// TIA Portal V20 export
FUNCTION_BLOCK "Sequence_20_Utility"   // FB240, LAD
AUTHOR : ERsystem_FA2_DH. Kim
// stored: IsIECCheckEnabled true, MemoryReserve 100, Namespace Unit1.Em6, SetENOAutomatically false
   VAR
      statSelectedJobNumber { ExternalWritable := 'False'} : DInt;   // Evaluated Job Number
      instSequenceLADStatus { ExternalWritable := 'False'} : "LAF_StatusLadSequence";
      instSequenceLADControl { ExternalWritable := 'False'} : "LAF_ControlLadSequence";
      statTonTime { ExternalAccessible := 'False'; ExternalVisible := 'False'; ExternalWritable := 'False'} : Array[0..999] of TON_TIME;
   END_VAR
   VAR CONSTANT
      STEP_IDLE : DInt := 1;
      STEP_IMMEDIATE_STOP : DInt := 9001;   // Step executed when an immediate stop command is triggered for the sequence (i.e. when unit is in state aborting)
      JOB_1_STEP_01 : DInt := 101;
      JOB_1_STEP_10 : DInt := 110;
      JOB_1_STEP_11 : DInt := 111;
      JOB_1_STEP_20 : DInt := 120;
      JOB_1_STEP_21 : DInt := 121;
      JOB_1_STEP_30 : DInt := 130;
      JOB_1_STEP_31 : DInt := 131;
      JOB_1_STEP_40 : DInt := 140;
      JOB_1_STEP_41 : DInt := 141;
      JOB_1_STEP_50 : DInt := 150;
      JOB_1_STEP_51 : DInt := 151;
      JOB_1_STEP_60 : DInt := 160;
      JOB_1_STEP_61 : DInt := 161;
      JOB_1_STEP_90 : DInt := 190;
      JOB_2_STEP_01 : DInt := 201;
      JOB_2_STEP_10 : DInt := 210;
      JOB_2_STEP_11 : DInt := 211;
      JOB_2_STEP_20 : DInt := 220;
      JOB_2_STEP_21 : DInt := 221;
      JOB_2_STEP_30 : DInt := 230;
      JOB_2_STEP_31 : DInt := 231;
      JOB_2_STEP_40 : DInt := 240;
      JOB_2_STEP_41 : DInt := 241;
      JOB_2_STEP_50 : DInt := 250;
      JOB_2_STEP_51 : DInt := 251;
      JOB_2_STEP_60 : DInt := 260;
      JOB_2_STEP_61 : DInt := 261;
      JOB_2_STEP_90 : DInt := 290;
   END_VAR
   VAR_TEMP   // added for the SCL form of the ladder/FBD networks
      _w1 : Bool;
   END_VAR
BEGIN

REGION Network 1: BLOCK INFO HEADER
   // (company) / (C) Copyright (year)
   // ---------------------------------------------------------------------------------
   // Title:                             (Title of this block)
   // Comment/Function: (that is implemented in the block)
   // Library/Family:           (that the source is dedicated to)
   // Author:                        (department / person in charge / contact)
   // Target System:          (test system with FW version)
   // Engineering:              TIA Portal (SW version)
   // Restrictions:               (OB types, etc.)
   // Requirements:           (hardware, technological package, etc.)
   // ---------------------------------------------------------------------------------
   // Change log table:
   // Version          | Date             | Signature      | Expert in charge  | Changes applied ------------------------|----------------------|-------------------------|--------------------------------|-----------------------
   // 001.000.000 | yyyy-mm-dd | 0x00000000 | (name of expert) | First released version
END_REGION

REGION Network 2: DESCRIPTION
   // This is a template block provided by the Automation Framework. It can be used to create an own project.
   // The Block Info Header is prepared to put in your own data.
   // Description of the block could be added here and the docu created by Code2Docu.
END_REGION

REGION Network 3: ********************* CONTROL *************************
END_REGION

REGION Network 4: Sequence Control
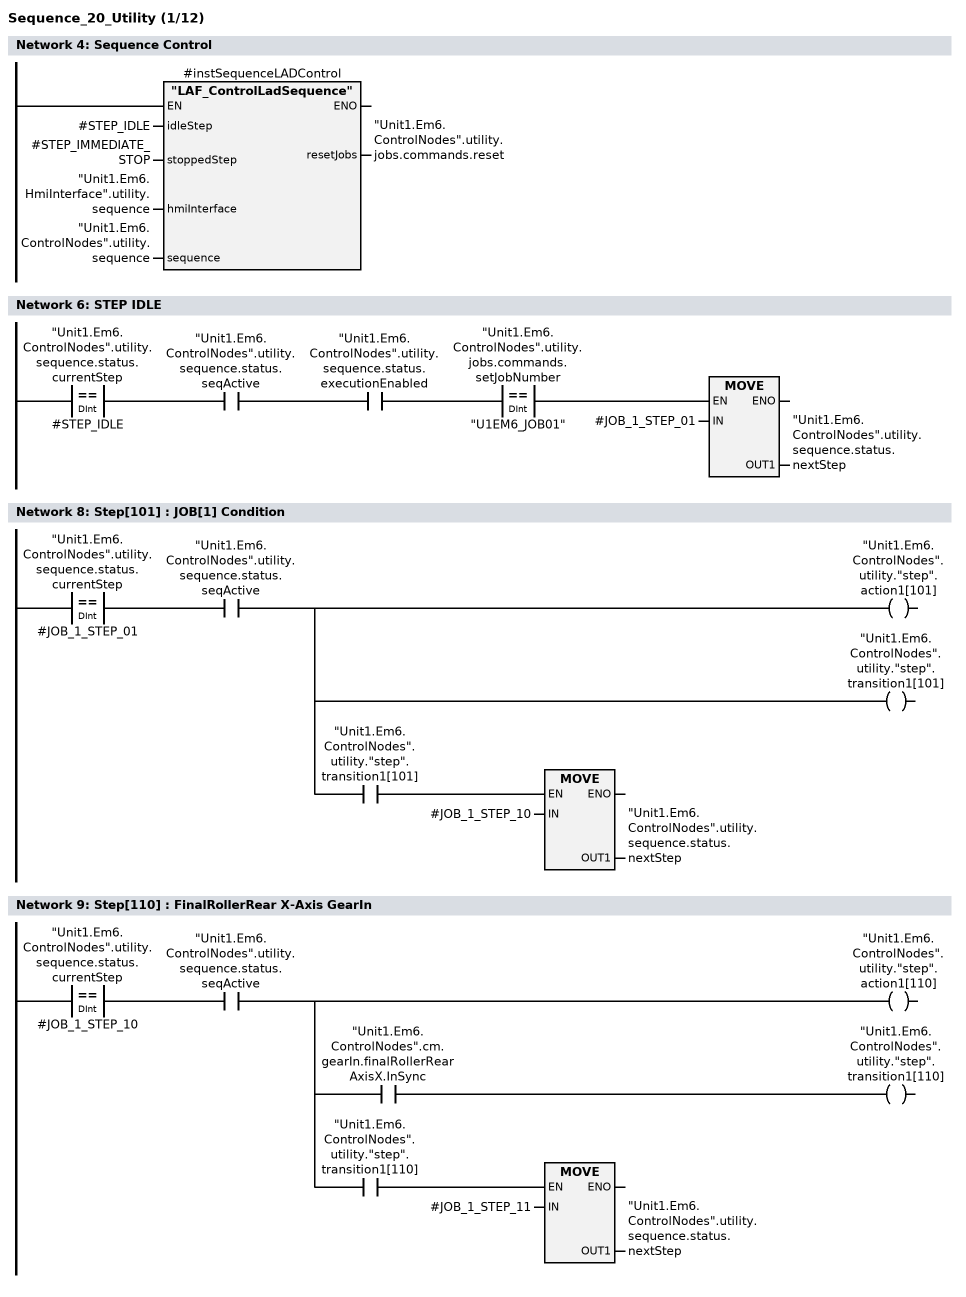
   RUNG wire#powerrail
      #instSequenceLADControl(idleStep := #STEP_IDLE, stoppedStep := #STEP_IMMEDIATE_STOP, hmiInterface := "Unit1.Em6.HmiInterface".utility.sequence, sequence := "Unit1.Em6.ControlNodes".utility.sequence, resetJobs => "Unit1.Em6.ControlNodes".utility.jobs.commands.reset)
   END_RUNG
   // the same network as SCL:
   #instSequenceLADControl(idleStep := #STEP_IDLE,   // "LAF_ControlLadSequence"
                           stoppedStep := #STEP_IMMEDIATE_STOP,
                           hmiInterface := "Unit1.Em6.HmiInterface".utility.sequence,
                           sequence := "Unit1.Em6.ControlNodes".utility.sequence,
                           resetJobs => "Unit1.Em6.ControlNodes".utility.jobs.commands.reset);
END_REGION

REGION Network 5: *************** JOB SELECT **************************
END_REGION

REGION Network 6: STEP IDLE
   RUNG wire#powerrail
      { S7_Templates := "SrcType := DInt" } EQ_Contact(in1 := "Unit1.Em6.ControlNodes".utility.sequence.status.currentStep, in2 := #STEP_IDLE)
      Contact( "Unit1.Em6.ControlNodes".utility.sequence.status.seqActive )
      Contact( "Unit1.Em6.ControlNodes".utility.sequence.status.executionEnabled )
      { S7_Templates := "SrcType := DInt" } EQ_Contact(in1 := "Unit1.Em6.ControlNodes".utility.jobs.commands.setJobNumber, in2 := "U1EM6_JOB01")
      Move(in := #JOB_1_STEP_01, out1 => "Unit1.Em6.ControlNodes".utility.sequence.status.nextStep)
   END_RUNG
   // the same network as SCL:
   IF ("Unit1.Em6.ControlNodes".utility.sequence.status.currentStep = #STEP_IDLE) AND "Unit1.Em6.ControlNodes".utility.sequence.status.seqActive AND "Unit1.Em6.ControlNodes".utility.sequence.status.executionEnabled AND ("Unit1.Em6.ControlNodes".utility.jobs.commands.setJobNumber = "U1EM6_JOB01") THEN
       "Unit1.Em6.ControlNodes".utility.sequence.status.nextStep := #JOB_1_STEP_01;
   END_IF;
END_REGION

REGION Network 7: *************** JOB[1] FinalRoller Gantry Home ************************
END_REGION

REGION Network 8: Step[101] : JOB[1] Condition
   RUNG wire#powerrail
      { S7_Templates := "SrcType := DInt" } EQ_Contact(in1 := "Unit1.Em6.ControlNodes".utility.sequence.status.currentStep, in2 := #JOB_1_STEP_01)
      Contact( "Unit1.Em6.ControlNodes".utility.sequence.status.seqActive )
      wire#w1
      Coil( "Unit1.Em6.ControlNodes".utility."step".action1[101] )
   END_RUNG
   RUNG wire#w1
      Coil( "Unit1.Em6.ControlNodes".utility."step".transition1[101] )
   END_RUNG
   RUNG wire#w1
      Contact( "Unit1.Em6.ControlNodes".utility."step".transition1[101] )
      Move(in := #JOB_1_STEP_10, out1 => "Unit1.Em6.ControlNodes".utility.sequence.status.nextStep)
   END_RUNG
   // the same network as SCL:
   "Unit1.Em6.ControlNodes".utility."step".action1[101] := ("Unit1.Em6.ControlNodes".utility.sequence.status.currentStep = #JOB_1_STEP_01) AND "Unit1.Em6.ControlNodes".utility.sequence.status.seqActive;
   "Unit1.Em6.ControlNodes".utility."step".transition1[101] := ("Unit1.Em6.ControlNodes".utility.sequence.status.currentStep = #JOB_1_STEP_01) AND "Unit1.Em6.ControlNodes".utility.sequence.status.seqActive;
   IF ("Unit1.Em6.ControlNodes".utility.sequence.status.currentStep = #JOB_1_STEP_01) AND "Unit1.Em6.ControlNodes".utility.sequence.status.seqActive AND "Unit1.Em6.ControlNodes".utility."step".transition1[101] THEN
       "Unit1.Em6.ControlNodes".utility.sequence.status.nextStep := #JOB_1_STEP_10;
   END_IF;
END_REGION

REGION Network 9: Step[110] : FinalRollerRear X-Axis GearIn
   RUNG wire#powerrail
      { S7_Templates := "SrcType := DInt" } EQ_Contact(in1 := "Unit1.Em6.ControlNodes".utility.sequence.status.currentStep, in2 := #JOB_1_STEP_10)
      Contact( "Unit1.Em6.ControlNodes".utility.sequence.status.seqActive )
      wire#w1
      Coil( "Unit1.Em6.ControlNodes".utility."step".action1[110] )
   END_RUNG
   RUNG wire#w1
      Contact( "Unit1.Em6.ControlNodes".cm.gearIn.finalRollerRearAxisX.InSync )
      Coil( "Unit1.Em6.ControlNodes".utility."step".transition1[110] )
   END_RUNG
   RUNG wire#w1
      Contact( "Unit1.Em6.ControlNodes".utility."step".transition1[110] )
      Move(in := #JOB_1_STEP_11, out1 => "Unit1.Em6.ControlNodes".utility.sequence.status.nextStep)
   END_RUNG
   // the same network as SCL:
   "Unit1.Em6.ControlNodes".utility."step".action1[110] := ("Unit1.Em6.ControlNodes".utility.sequence.status.currentStep = #JOB_1_STEP_10) AND "Unit1.Em6.ControlNodes".utility.sequence.status.seqActive;
   "Unit1.Em6.ControlNodes".utility."step".transition1[110] := ("Unit1.Em6.ControlNodes".utility.sequence.status.currentStep = #JOB_1_STEP_10) AND "Unit1.Em6.ControlNodes".utility.sequence.status.seqActive AND "Unit1.Em6.ControlNodes".cm.gearIn.finalRollerRearAxisX.InSync;
   IF ("Unit1.Em6.ControlNodes".utility.sequence.status.currentStep = #JOB_1_STEP_10) AND "Unit1.Em6.ControlNodes".utility.sequence.status.seqActive AND "Unit1.Em6.ControlNodes".utility."step".transition1[110] THEN
       "Unit1.Em6.ControlNodes".utility.sequence.status.nextStep := #JOB_1_STEP_11;
   END_IF;
END_REGION

REGION Network 10: Step[111] : FinalRollerRear X-Axis LimitSensor Off
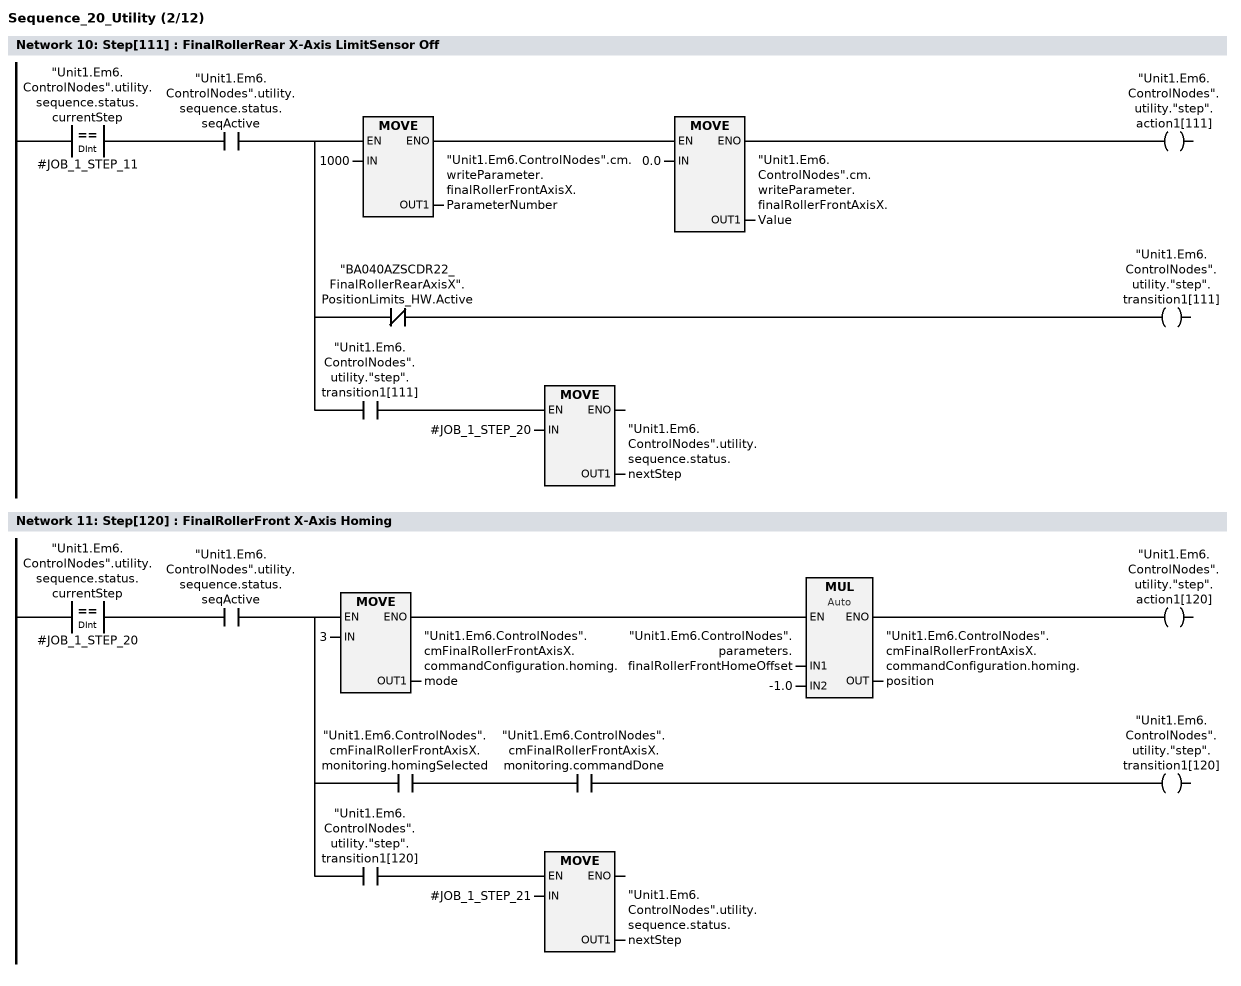
   RUNG wire#powerrail
      { S7_Templates := "SrcType := DInt" } EQ_Contact(in1 := "Unit1.Em6.ControlNodes".utility.sequence.status.currentStep, in2 := #JOB_1_STEP_11)
      Contact( "Unit1.Em6.ControlNodes".utility.sequence.status.seqActive )
      wire#w1
      Move(in := 1000, out1 => "Unit1.Em6.ControlNodes".cm.writeParameter.finalRollerFrontAxisX.ParameterNumber)
      Move(in := 0.0, out1 => "Unit1.Em6.ControlNodes".cm.writeParameter.finalRollerFrontAxisX.Value)
      Coil( "Unit1.Em6.ControlNodes".utility."step".action1[111] )
   END_RUNG
   RUNG wire#w1
      I_Contact( "BA040AZSCDR22_FinalRollerRearAxisX".PositionLimits_HW.Active )
      Coil( "Unit1.Em6.ControlNodes".utility."step".transition1[111] )
   END_RUNG
   RUNG wire#w1
      Contact( "Unit1.Em6.ControlNodes".utility."step".transition1[111] )
      Move(in := #JOB_1_STEP_20, out1 => "Unit1.Em6.ControlNodes".utility.sequence.status.nextStep)
   END_RUNG
   // the same network as SCL:
   #_w1 := ("Unit1.Em6.ControlNodes".utility.sequence.status.currentStep = #JOB_1_STEP_11) AND "Unit1.Em6.ControlNodes".utility.sequence.status.seqActive;
   IF #_w1 THEN
       "Unit1.Em6.ControlNodes".cm.writeParameter.finalRollerFrontAxisX.ParameterNumber := 1000;
       "Unit1.Em6.ControlNodes".cm.writeParameter.finalRollerFrontAxisX.Value := 0.0;
   END_IF;
   "Unit1.Em6.ControlNodes".utility."step".action1[111] := #_w1;
   "Unit1.Em6.ControlNodes".utility."step".transition1[111] := #_w1 AND NOT "BA040AZSCDR22_FinalRollerRearAxisX".PositionLimits_HW.Active;
   IF #_w1 AND "Unit1.Em6.ControlNodes".utility."step".transition1[111] THEN
       "Unit1.Em6.ControlNodes".utility.sequence.status.nextStep := #JOB_1_STEP_20;
   END_IF;
END_REGION

REGION Network 11: Step[120] : FinalRollerFront X-Axis Homing
   RUNG wire#powerrail
      { S7_Templates := "SrcType := DInt" } EQ_Contact(in1 := "Unit1.Em6.ControlNodes".utility.sequence.status.currentStep, in2 := #JOB_1_STEP_20)
      Contact( "Unit1.Em6.ControlNodes".utility.sequence.status.seqActive )
      wire#w1
      Move(in := 3, out1 => "Unit1.Em6.ControlNodes".cmFinalRollerFrontAxisX.commandConfiguration.homing.mode)
      Mul(in1 := "Unit1.Em6.ControlNodes".parameters.finalRollerFrontHomeOffset, in2 := -1.0, out => "Unit1.Em6.ControlNodes".cmFinalRollerFrontAxisX.commandConfiguration.homing.position)
      Coil( "Unit1.Em6.ControlNodes".utility."step".action1[120] )
   END_RUNG
   RUNG wire#w1
      Contact( "Unit1.Em6.ControlNodes".cmFinalRollerFrontAxisX.monitoring.homingSelected )
      Contact( "Unit1.Em6.ControlNodes".cmFinalRollerFrontAxisX.monitoring.commandDone )
      Coil( "Unit1.Em6.ControlNodes".utility."step".transition1[120] )
   END_RUNG
   RUNG wire#w1
      Contact( "Unit1.Em6.ControlNodes".utility."step".transition1[120] )
      Move(in := #JOB_1_STEP_21, out1 => "Unit1.Em6.ControlNodes".utility.sequence.status.nextStep)
   END_RUNG
   // the same network as SCL:
   #_w1 := ("Unit1.Em6.ControlNodes".utility.sequence.status.currentStep = #JOB_1_STEP_20) AND "Unit1.Em6.ControlNodes".utility.sequence.status.seqActive;
   IF #_w1 THEN
       "Unit1.Em6.ControlNodes".cmFinalRollerFrontAxisX.commandConfiguration.homing.mode := 3;
       "Unit1.Em6.ControlNodes".cmFinalRollerFrontAxisX.commandConfiguration.homing.position := "Unit1.Em6.ControlNodes".parameters.finalRollerFrontHomeOffset * (-1.0);
   END_IF;
   "Unit1.Em6.ControlNodes".utility."step".action1[120] := #_w1;
   "Unit1.Em6.ControlNodes".utility."step".transition1[120] := #_w1 AND "Unit1.Em6.ControlNodes".cmFinalRollerFrontAxisX.monitoring.homingSelected AND "Unit1.Em6.ControlNodes".cmFinalRollerFrontAxisX.monitoring.commandDone;
   IF #_w1 AND "Unit1.Em6.ControlNodes".utility."step".transition1[120] THEN
       "Unit1.Em6.ControlNodes".utility.sequence.status.nextStep := #JOB_1_STEP_21;
   END_IF;
END_REGION

REGION Network 12: Step[121] : FinalRollerFront X-Axis Move Home
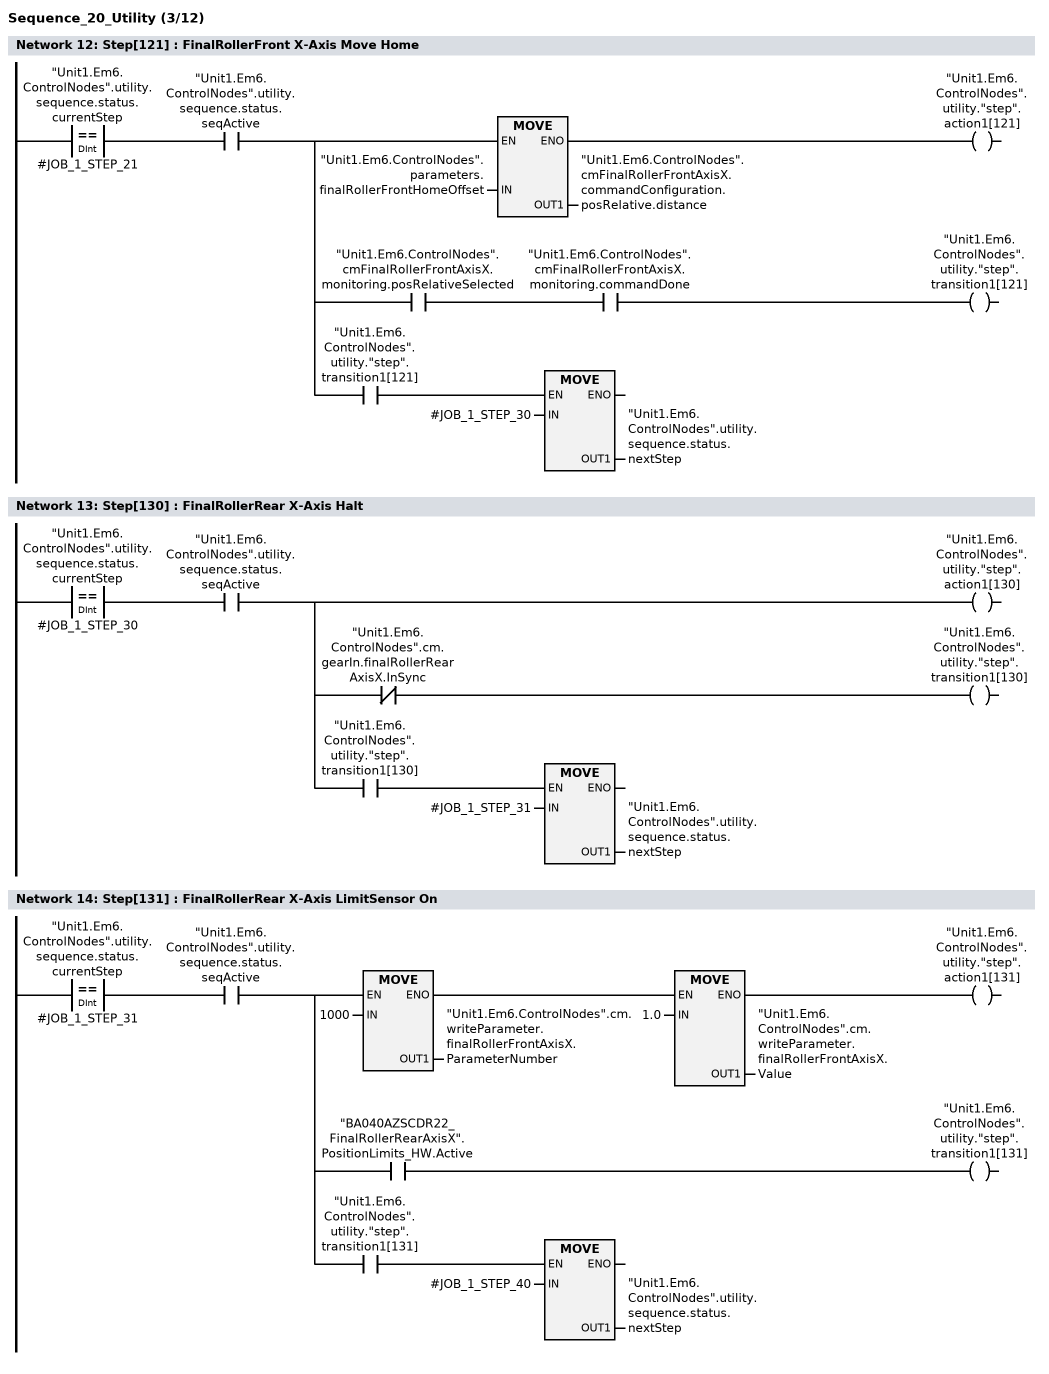
   RUNG wire#powerrail
      { S7_Templates := "SrcType := DInt" } EQ_Contact(in1 := "Unit1.Em6.ControlNodes".utility.sequence.status.currentStep, in2 := #JOB_1_STEP_21)
      Contact( "Unit1.Em6.ControlNodes".utility.sequence.status.seqActive )
      wire#w1
      Move(in := "Unit1.Em6.ControlNodes".parameters.finalRollerFrontHomeOffset, out1 => "Unit1.Em6.ControlNodes".cmFinalRollerFrontAxisX.commandConfiguration.posRelative.distance)
      Coil( "Unit1.Em6.ControlNodes".utility."step".action1[121] )
   END_RUNG
   RUNG wire#w1
      Contact( "Unit1.Em6.ControlNodes".cmFinalRollerFrontAxisX.monitoring.posRelativeSelected )
      Contact( "Unit1.Em6.ControlNodes".cmFinalRollerFrontAxisX.monitoring.commandDone )
      Coil( "Unit1.Em6.ControlNodes".utility."step".transition1[121] )
   END_RUNG
   RUNG wire#w1
      Contact( "Unit1.Em6.ControlNodes".utility."step".transition1[121] )
      Move(in := #JOB_1_STEP_30, out1 => "Unit1.Em6.ControlNodes".utility.sequence.status.nextStep)
   END_RUNG
   // the same network as SCL:
   #_w1 := ("Unit1.Em6.ControlNodes".utility.sequence.status.currentStep = #JOB_1_STEP_21) AND "Unit1.Em6.ControlNodes".utility.sequence.status.seqActive;
   IF #_w1 THEN
       "Unit1.Em6.ControlNodes".cmFinalRollerFrontAxisX.commandConfiguration.posRelative.distance := "Unit1.Em6.ControlNodes".parameters.finalRollerFrontHomeOffset;
   END_IF;
   "Unit1.Em6.ControlNodes".utility."step".action1[121] := #_w1;
   "Unit1.Em6.ControlNodes".utility."step".transition1[121] := #_w1 AND "Unit1.Em6.ControlNodes".cmFinalRollerFrontAxisX.monitoring.posRelativeSelected AND "Unit1.Em6.ControlNodes".cmFinalRollerFrontAxisX.monitoring.commandDone;
   IF #_w1 AND "Unit1.Em6.ControlNodes".utility."step".transition1[121] THEN
       "Unit1.Em6.ControlNodes".utility.sequence.status.nextStep := #JOB_1_STEP_30;
   END_IF;
END_REGION

REGION Network 13: Step[130] : FinalRollerRear X-Axis Halt
   RUNG wire#powerrail
      { S7_Templates := "SrcType := DInt" } EQ_Contact(in1 := "Unit1.Em6.ControlNodes".utility.sequence.status.currentStep, in2 := #JOB_1_STEP_30)
      Contact( "Unit1.Em6.ControlNodes".utility.sequence.status.seqActive )
      wire#w1
      Coil( "Unit1.Em6.ControlNodes".utility."step".action1[130] )
   END_RUNG
   RUNG wire#w1
      I_Contact( "Unit1.Em6.ControlNodes".cm.gearIn.finalRollerRearAxisX.InSync )
      Coil( "Unit1.Em6.ControlNodes".utility."step".transition1[130] )
   END_RUNG
   RUNG wire#w1
      Contact( "Unit1.Em6.ControlNodes".utility."step".transition1[130] )
      Move(in := #JOB_1_STEP_31, out1 => "Unit1.Em6.ControlNodes".utility.sequence.status.nextStep)
   END_RUNG
   // the same network as SCL:
   "Unit1.Em6.ControlNodes".utility."step".action1[130] := ("Unit1.Em6.ControlNodes".utility.sequence.status.currentStep = #JOB_1_STEP_30) AND "Unit1.Em6.ControlNodes".utility.sequence.status.seqActive;
   "Unit1.Em6.ControlNodes".utility."step".transition1[130] := ("Unit1.Em6.ControlNodes".utility.sequence.status.currentStep = #JOB_1_STEP_30) AND "Unit1.Em6.ControlNodes".utility.sequence.status.seqActive AND NOT "Unit1.Em6.ControlNodes".cm.gearIn.finalRollerRearAxisX.InSync;
   IF ("Unit1.Em6.ControlNodes".utility.sequence.status.currentStep = #JOB_1_STEP_30) AND "Unit1.Em6.ControlNodes".utility.sequence.status.seqActive AND "Unit1.Em6.ControlNodes".utility."step".transition1[130] THEN
       "Unit1.Em6.ControlNodes".utility.sequence.status.nextStep := #JOB_1_STEP_31;
   END_IF;
END_REGION

REGION Network 14: Step[131] : FinalRollerRear X-Axis LimitSensor On
   RUNG wire#powerrail
      { S7_Templates := "SrcType := DInt" } EQ_Contact(in1 := "Unit1.Em6.ControlNodes".utility.sequence.status.currentStep, in2 := #JOB_1_STEP_31)
      Contact( "Unit1.Em6.ControlNodes".utility.sequence.status.seqActive )
      wire#w1
      Move(in := 1000, out1 => "Unit1.Em6.ControlNodes".cm.writeParameter.finalRollerFrontAxisX.ParameterNumber)
      Move(in := 1.0, out1 => "Unit1.Em6.ControlNodes".cm.writeParameter.finalRollerFrontAxisX.Value)
      Coil( "Unit1.Em6.ControlNodes".utility."step".action1[131] )
   END_RUNG
   RUNG wire#w1
      Contact( "BA040AZSCDR22_FinalRollerRearAxisX".PositionLimits_HW.Active )
      Coil( "Unit1.Em6.ControlNodes".utility."step".transition1[131] )
   END_RUNG
   RUNG wire#w1
      Contact( "Unit1.Em6.ControlNodes".utility."step".transition1[131] )
      Move(in := #JOB_1_STEP_40, out1 => "Unit1.Em6.ControlNodes".utility.sequence.status.nextStep)
   END_RUNG
   // the same network as SCL:
   #_w1 := ("Unit1.Em6.ControlNodes".utility.sequence.status.currentStep = #JOB_1_STEP_31) AND "Unit1.Em6.ControlNodes".utility.sequence.status.seqActive;
   IF #_w1 THEN
       "Unit1.Em6.ControlNodes".cm.writeParameter.finalRollerFrontAxisX.ParameterNumber := 1000;
       "Unit1.Em6.ControlNodes".cm.writeParameter.finalRollerFrontAxisX.Value := 1.0;
   END_IF;
   "Unit1.Em6.ControlNodes".utility."step".action1[131] := #_w1;
   "Unit1.Em6.ControlNodes".utility."step".transition1[131] := #_w1 AND "BA040AZSCDR22_FinalRollerRearAxisX".PositionLimits_HW.Active;
   IF #_w1 AND "Unit1.Em6.ControlNodes".utility."step".transition1[131] THEN
       "Unit1.Em6.ControlNodes".utility.sequence.status.nextStep := #JOB_1_STEP_40;
   END_IF;
END_REGION

REGION Network 15: Step[140] : FinalRollerFront X-Axis GearIn
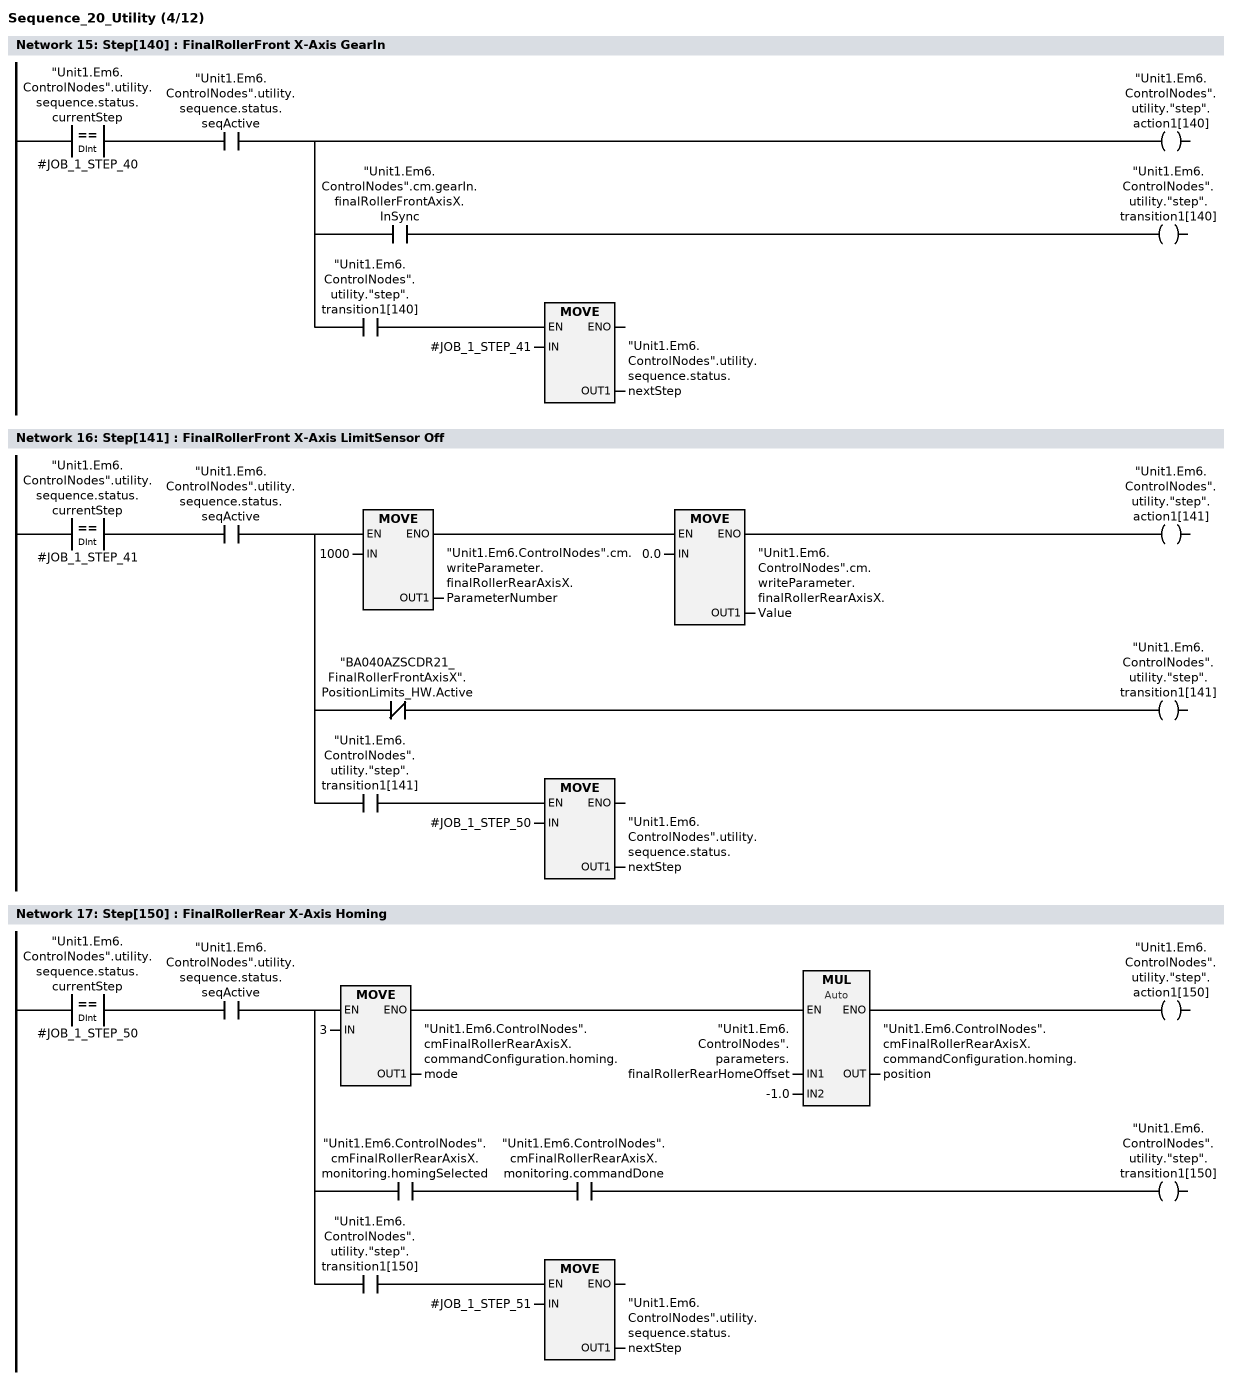
   RUNG wire#powerrail
      { S7_Templates := "SrcType := DInt" } EQ_Contact(in1 := "Unit1.Em6.ControlNodes".utility.sequence.status.currentStep, in2 := #JOB_1_STEP_40)
      Contact( "Unit1.Em6.ControlNodes".utility.sequence.status.seqActive )
      wire#w1
      Coil( "Unit1.Em6.ControlNodes".utility."step".action1[140] )
   END_RUNG
   RUNG wire#w1
      Contact( "Unit1.Em6.ControlNodes".cm.gearIn.finalRollerFrontAxisX.InSync )
      Coil( "Unit1.Em6.ControlNodes".utility."step".transition1[140] )
   END_RUNG
   RUNG wire#w1
      Contact( "Unit1.Em6.ControlNodes".utility."step".transition1[140] )
      Move(in := #JOB_1_STEP_41, out1 => "Unit1.Em6.ControlNodes".utility.sequence.status.nextStep)
   END_RUNG
   // the same network as SCL:
   "Unit1.Em6.ControlNodes".utility."step".action1[140] := ("Unit1.Em6.ControlNodes".utility.sequence.status.currentStep = #JOB_1_STEP_40) AND "Unit1.Em6.ControlNodes".utility.sequence.status.seqActive;
   "Unit1.Em6.ControlNodes".utility."step".transition1[140] := ("Unit1.Em6.ControlNodes".utility.sequence.status.currentStep = #JOB_1_STEP_40) AND "Unit1.Em6.ControlNodes".utility.sequence.status.seqActive AND "Unit1.Em6.ControlNodes".cm.gearIn.finalRollerFrontAxisX.InSync;
   IF ("Unit1.Em6.ControlNodes".utility.sequence.status.currentStep = #JOB_1_STEP_40) AND "Unit1.Em6.ControlNodes".utility.sequence.status.seqActive AND "Unit1.Em6.ControlNodes".utility."step".transition1[140] THEN
       "Unit1.Em6.ControlNodes".utility.sequence.status.nextStep := #JOB_1_STEP_41;
   END_IF;
END_REGION

REGION Network 16: Step[141] : FinalRollerFront X-Axis LimitSensor Off
   RUNG wire#powerrail
      { S7_Templates := "SrcType := DInt" } EQ_Contact(in1 := "Unit1.Em6.ControlNodes".utility.sequence.status.currentStep, in2 := #JOB_1_STEP_41)
      Contact( "Unit1.Em6.ControlNodes".utility.sequence.status.seqActive )
      wire#w1
      Move(in := 1000, out1 => "Unit1.Em6.ControlNodes".cm.writeParameter.finalRollerRearAxisX.ParameterNumber)
      Move(in := 0.0, out1 => "Unit1.Em6.ControlNodes".cm.writeParameter.finalRollerRearAxisX.Value)
      Coil( "Unit1.Em6.ControlNodes".utility."step".action1[141] )
   END_RUNG
   RUNG wire#w1
      I_Contact( "BA040AZSCDR21_FinalRollerFrontAxisX".PositionLimits_HW.Active )
      Coil( "Unit1.Em6.ControlNodes".utility."step".transition1[141] )
   END_RUNG
   RUNG wire#w1
      Contact( "Unit1.Em6.ControlNodes".utility."step".transition1[141] )
      Move(in := #JOB_1_STEP_50, out1 => "Unit1.Em6.ControlNodes".utility.sequence.status.nextStep)
   END_RUNG
   // the same network as SCL:
   #_w1 := ("Unit1.Em6.ControlNodes".utility.sequence.status.currentStep = #JOB_1_STEP_41) AND "Unit1.Em6.ControlNodes".utility.sequence.status.seqActive;
   IF #_w1 THEN
       "Unit1.Em6.ControlNodes".cm.writeParameter.finalRollerRearAxisX.ParameterNumber := 1000;
       "Unit1.Em6.ControlNodes".cm.writeParameter.finalRollerRearAxisX.Value := 0.0;
   END_IF;
   "Unit1.Em6.ControlNodes".utility."step".action1[141] := #_w1;
   "Unit1.Em6.ControlNodes".utility."step".transition1[141] := #_w1 AND NOT "BA040AZSCDR21_FinalRollerFrontAxisX".PositionLimits_HW.Active;
   IF #_w1 AND "Unit1.Em6.ControlNodes".utility."step".transition1[141] THEN
       "Unit1.Em6.ControlNodes".utility.sequence.status.nextStep := #JOB_1_STEP_50;
   END_IF;
END_REGION

REGION Network 17: Step[150] : FinalRollerRear X-Axis Homing
   RUNG wire#powerrail
      { S7_Templates := "SrcType := DInt" } EQ_Contact(in1 := "Unit1.Em6.ControlNodes".utility.sequence.status.currentStep, in2 := #JOB_1_STEP_50)
      Contact( "Unit1.Em6.ControlNodes".utility.sequence.status.seqActive )
      wire#w1
      Move(in := 3, out1 => "Unit1.Em6.ControlNodes".cmFinalRollerRearAxisX.commandConfiguration.homing.mode)
      Mul(in1 := "Unit1.Em6.ControlNodes".parameters.finalRollerRearHomeOffset, in2 := -1.0, out => "Unit1.Em6.ControlNodes".cmFinalRollerRearAxisX.commandConfiguration.homing.position)
      Coil( "Unit1.Em6.ControlNodes".utility."step".action1[150] )
   END_RUNG
   RUNG wire#w1
      Contact( "Unit1.Em6.ControlNodes".cmFinalRollerRearAxisX.monitoring.homingSelected )
      Contact( "Unit1.Em6.ControlNodes".cmFinalRollerRearAxisX.monitoring.commandDone )
      Coil( "Unit1.Em6.ControlNodes".utility."step".transition1[150] )
   END_RUNG
   RUNG wire#w1
      Contact( "Unit1.Em6.ControlNodes".utility."step".transition1[150] )
      Move(in := #JOB_1_STEP_51, out1 => "Unit1.Em6.ControlNodes".utility.sequence.status.nextStep)
   END_RUNG
   // the same network as SCL:
   #_w1 := ("Unit1.Em6.ControlNodes".utility.sequence.status.currentStep = #JOB_1_STEP_50) AND "Unit1.Em6.ControlNodes".utility.sequence.status.seqActive;
   IF #_w1 THEN
       "Unit1.Em6.ControlNodes".cmFinalRollerRearAxisX.commandConfiguration.homing.mode := 3;
       "Unit1.Em6.ControlNodes".cmFinalRollerRearAxisX.commandConfiguration.homing.position := "Unit1.Em6.ControlNodes".parameters.finalRollerRearHomeOffset * (-1.0);
   END_IF;
   "Unit1.Em6.ControlNodes".utility."step".action1[150] := #_w1;
   "Unit1.Em6.ControlNodes".utility."step".transition1[150] := #_w1 AND "Unit1.Em6.ControlNodes".cmFinalRollerRearAxisX.monitoring.homingSelected AND "Unit1.Em6.ControlNodes".cmFinalRollerRearAxisX.monitoring.commandDone;
   IF #_w1 AND "Unit1.Em6.ControlNodes".utility."step".transition1[150] THEN
       "Unit1.Em6.ControlNodes".utility.sequence.status.nextStep := #JOB_1_STEP_51;
   END_IF;
END_REGION

REGION Network 18: Step[151] : FinalRollerRear X-Axis Move Home
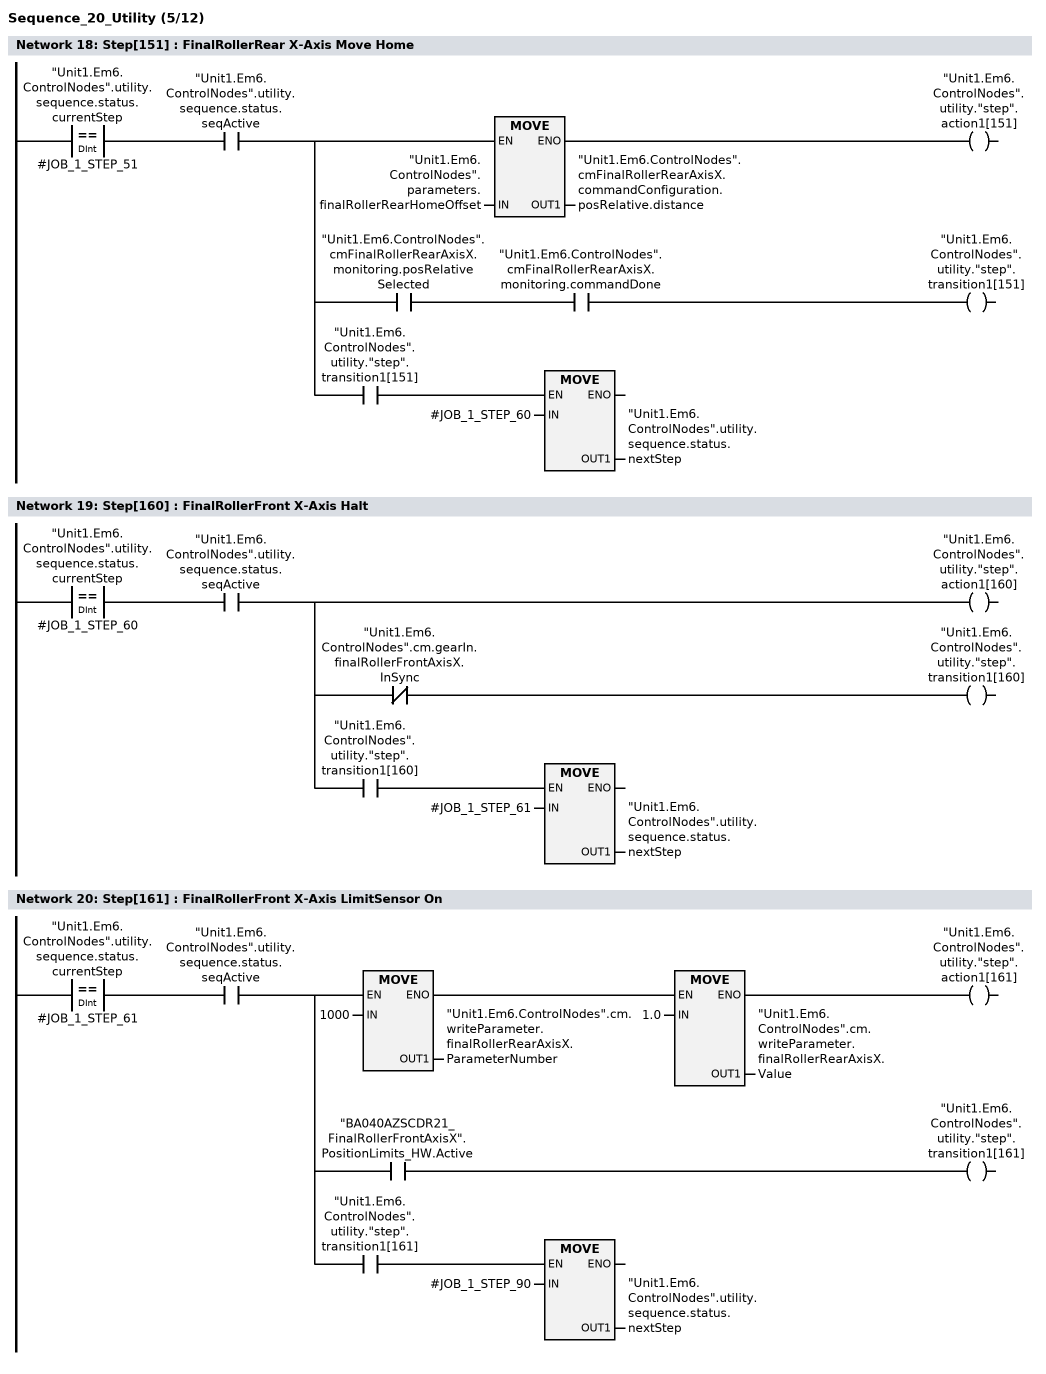
   RUNG wire#powerrail
      { S7_Templates := "SrcType := DInt" } EQ_Contact(in1 := "Unit1.Em6.ControlNodes".utility.sequence.status.currentStep, in2 := #JOB_1_STEP_51)
      Contact( "Unit1.Em6.ControlNodes".utility.sequence.status.seqActive )
      wire#w1
      Move(in := "Unit1.Em6.ControlNodes".parameters.finalRollerRearHomeOffset, out1 => "Unit1.Em6.ControlNodes".cmFinalRollerRearAxisX.commandConfiguration.posRelative.distance)
      Coil( "Unit1.Em6.ControlNodes".utility."step".action1[151] )
   END_RUNG
   RUNG wire#w1
      Contact( "Unit1.Em6.ControlNodes".cmFinalRollerRearAxisX.monitoring.posRelativeSelected )
      Contact( "Unit1.Em6.ControlNodes".cmFinalRollerRearAxisX.monitoring.commandDone )
      Coil( "Unit1.Em6.ControlNodes".utility."step".transition1[151] )
   END_RUNG
   RUNG wire#w1
      Contact( "Unit1.Em6.ControlNodes".utility."step".transition1[151] )
      Move(in := #JOB_1_STEP_60, out1 => "Unit1.Em6.ControlNodes".utility.sequence.status.nextStep)
   END_RUNG
   // the same network as SCL:
   #_w1 := ("Unit1.Em6.ControlNodes".utility.sequence.status.currentStep = #JOB_1_STEP_51) AND "Unit1.Em6.ControlNodes".utility.sequence.status.seqActive;
   IF #_w1 THEN
       "Unit1.Em6.ControlNodes".cmFinalRollerRearAxisX.commandConfiguration.posRelative.distance := "Unit1.Em6.ControlNodes".parameters.finalRollerRearHomeOffset;
   END_IF;
   "Unit1.Em6.ControlNodes".utility."step".action1[151] := #_w1;
   "Unit1.Em6.ControlNodes".utility."step".transition1[151] := #_w1 AND "Unit1.Em6.ControlNodes".cmFinalRollerRearAxisX.monitoring.posRelativeSelected AND "Unit1.Em6.ControlNodes".cmFinalRollerRearAxisX.monitoring.commandDone;
   IF #_w1 AND "Unit1.Em6.ControlNodes".utility."step".transition1[151] THEN
       "Unit1.Em6.ControlNodes".utility.sequence.status.nextStep := #JOB_1_STEP_60;
   END_IF;
END_REGION

REGION Network 19: Step[160] : FinalRollerFront X-Axis Halt
   RUNG wire#powerrail
      { S7_Templates := "SrcType := DInt" } EQ_Contact(in1 := "Unit1.Em6.ControlNodes".utility.sequence.status.currentStep, in2 := #JOB_1_STEP_60)
      Contact( "Unit1.Em6.ControlNodes".utility.sequence.status.seqActive )
      wire#w1
      Coil( "Unit1.Em6.ControlNodes".utility."step".action1[160] )
   END_RUNG
   RUNG wire#w1
      I_Contact( "Unit1.Em6.ControlNodes".cm.gearIn.finalRollerFrontAxisX.InSync )
      Coil( "Unit1.Em6.ControlNodes".utility."step".transition1[160] )
   END_RUNG
   RUNG wire#w1
      Contact( "Unit1.Em6.ControlNodes".utility."step".transition1[160] )
      Move(in := #JOB_1_STEP_61, out1 => "Unit1.Em6.ControlNodes".utility.sequence.status.nextStep)
   END_RUNG
   // the same network as SCL:
   "Unit1.Em6.ControlNodes".utility."step".action1[160] := ("Unit1.Em6.ControlNodes".utility.sequence.status.currentStep = #JOB_1_STEP_60) AND "Unit1.Em6.ControlNodes".utility.sequence.status.seqActive;
   "Unit1.Em6.ControlNodes".utility."step".transition1[160] := ("Unit1.Em6.ControlNodes".utility.sequence.status.currentStep = #JOB_1_STEP_60) AND "Unit1.Em6.ControlNodes".utility.sequence.status.seqActive AND NOT "Unit1.Em6.ControlNodes".cm.gearIn.finalRollerFrontAxisX.InSync;
   IF ("Unit1.Em6.ControlNodes".utility.sequence.status.currentStep = #JOB_1_STEP_60) AND "Unit1.Em6.ControlNodes".utility.sequence.status.seqActive AND "Unit1.Em6.ControlNodes".utility."step".transition1[160] THEN
       "Unit1.Em6.ControlNodes".utility.sequence.status.nextStep := #JOB_1_STEP_61;
   END_IF;
END_REGION

REGION Network 20: Step[161] : FinalRollerFront X-Axis LimitSensor On
   RUNG wire#powerrail
      { S7_Templates := "SrcType := DInt" } EQ_Contact(in1 := "Unit1.Em6.ControlNodes".utility.sequence.status.currentStep, in2 := #JOB_1_STEP_61)
      Contact( "Unit1.Em6.ControlNodes".utility.sequence.status.seqActive )
      wire#w1
      Move(in := 1000, out1 => "Unit1.Em6.ControlNodes".cm.writeParameter.finalRollerRearAxisX.ParameterNumber)
      Move(in := 1.0, out1 => "Unit1.Em6.ControlNodes".cm.writeParameter.finalRollerRearAxisX.Value)
      Coil( "Unit1.Em6.ControlNodes".utility."step".action1[161] )
   END_RUNG
   RUNG wire#w1
      Contact( "BA040AZSCDR21_FinalRollerFrontAxisX".PositionLimits_HW.Active )
      Coil( "Unit1.Em6.ControlNodes".utility."step".transition1[161] )
   END_RUNG
   RUNG wire#w1
      Contact( "Unit1.Em6.ControlNodes".utility."step".transition1[161] )
      Move(in := #JOB_1_STEP_90, out1 => "Unit1.Em6.ControlNodes".utility.sequence.status.nextStep)
   END_RUNG
   // the same network as SCL:
   #_w1 := ("Unit1.Em6.ControlNodes".utility.sequence.status.currentStep = #JOB_1_STEP_61) AND "Unit1.Em6.ControlNodes".utility.sequence.status.seqActive;
   IF #_w1 THEN
       "Unit1.Em6.ControlNodes".cm.writeParameter.finalRollerRearAxisX.ParameterNumber := 1000;
       "Unit1.Em6.ControlNodes".cm.writeParameter.finalRollerRearAxisX.Value := 1.0;
   END_IF;
   "Unit1.Em6.ControlNodes".utility."step".action1[161] := #_w1;
   "Unit1.Em6.ControlNodes".utility."step".transition1[161] := #_w1 AND "BA040AZSCDR21_FinalRollerFrontAxisX".PositionLimits_HW.Active;
   IF #_w1 AND "Unit1.Em6.ControlNodes".utility."step".transition1[161] THEN
       "Unit1.Em6.ControlNodes".utility.sequence.status.nextStep := #JOB_1_STEP_90;
   END_IF;
END_REGION

REGION Network 21: Step[190] : JOB[1] Step End
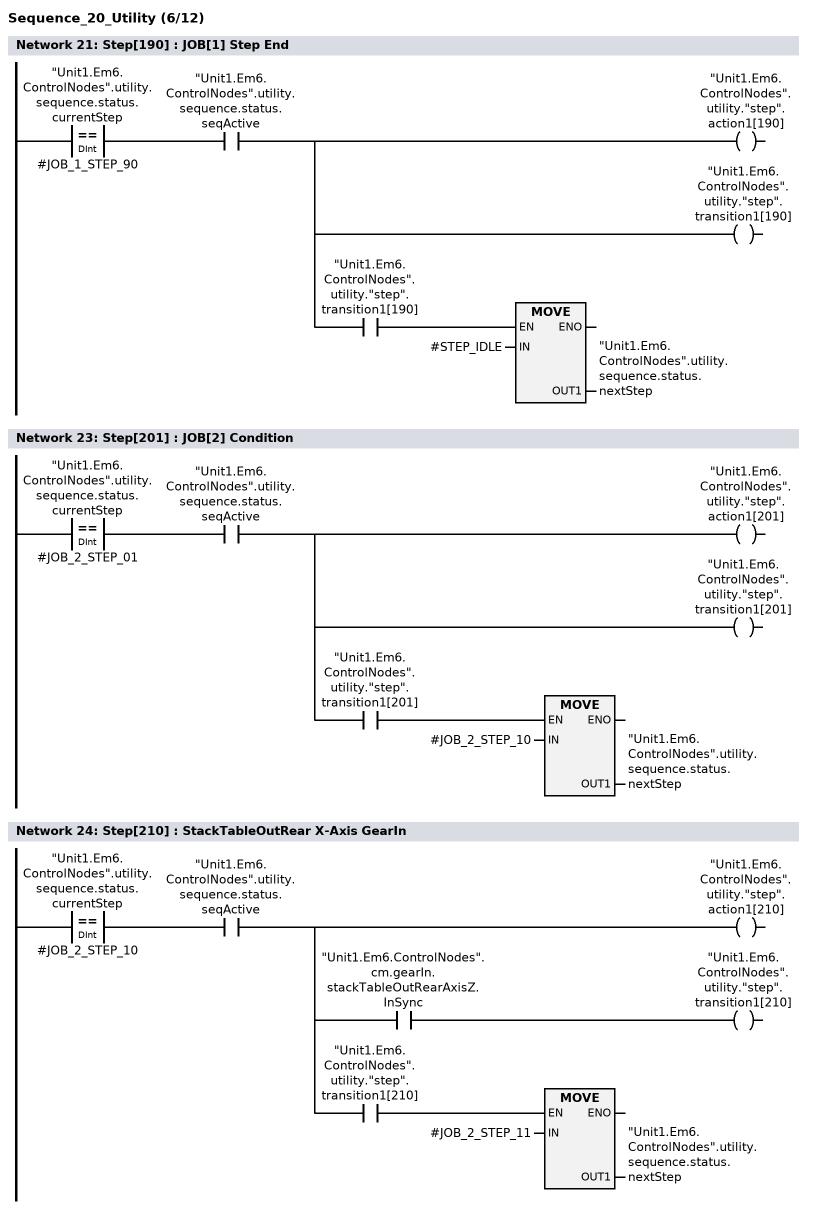
   RUNG wire#powerrail
      { S7_Templates := "SrcType := DInt" } EQ_Contact(in1 := "Unit1.Em6.ControlNodes".utility.sequence.status.currentStep, in2 := #JOB_1_STEP_90)
      Contact( "Unit1.Em6.ControlNodes".utility.sequence.status.seqActive )
      wire#w1
      Coil( "Unit1.Em6.ControlNodes".utility."step".action1[190] )
   END_RUNG
   RUNG wire#w1
      Coil( "Unit1.Em6.ControlNodes".utility."step".transition1[190] )
   END_RUNG
   RUNG wire#w1
      Contact( "Unit1.Em6.ControlNodes".utility."step".transition1[190] )
      Move(in := #STEP_IDLE, out1 => "Unit1.Em6.ControlNodes".utility.sequence.status.nextStep)
   END_RUNG
   // the same network as SCL:
   "Unit1.Em6.ControlNodes".utility."step".action1[190] := ("Unit1.Em6.ControlNodes".utility.sequence.status.currentStep = #JOB_1_STEP_90) AND "Unit1.Em6.ControlNodes".utility.sequence.status.seqActive;
   "Unit1.Em6.ControlNodes".utility."step".transition1[190] := ("Unit1.Em6.ControlNodes".utility.sequence.status.currentStep = #JOB_1_STEP_90) AND "Unit1.Em6.ControlNodes".utility.sequence.status.seqActive;
   IF ("Unit1.Em6.ControlNodes".utility.sequence.status.currentStep = #JOB_1_STEP_90) AND "Unit1.Em6.ControlNodes".utility.sequence.status.seqActive AND "Unit1.Em6.ControlNodes".utility."step".transition1[190] THEN
       "Unit1.Em6.ControlNodes".utility.sequence.status.nextStep := #STEP_IDLE;
   END_IF;
END_REGION

REGION Network 22: *************** JOB[2] StackTableOut Gantry Home ************************
END_REGION

REGION Network 23: Step[201] : JOB[2] Condition
   RUNG wire#powerrail
      { S7_Templates := "SrcType := DInt" } EQ_Contact(in1 := "Unit1.Em6.ControlNodes".utility.sequence.status.currentStep, in2 := #JOB_2_STEP_01)
      Contact( "Unit1.Em6.ControlNodes".utility.sequence.status.seqActive )
      wire#w1
      Coil( "Unit1.Em6.ControlNodes".utility."step".action1[201] )
   END_RUNG
   RUNG wire#w1
      Coil( "Unit1.Em6.ControlNodes".utility."step".transition1[201] )
   END_RUNG
   RUNG wire#w1
      Contact( "Unit1.Em6.ControlNodes".utility."step".transition1[201] )
      Move(in := #JOB_2_STEP_10, out1 => "Unit1.Em6.ControlNodes".utility.sequence.status.nextStep)
   END_RUNG
   // the same network as SCL:
   "Unit1.Em6.ControlNodes".utility."step".action1[201] := ("Unit1.Em6.ControlNodes".utility.sequence.status.currentStep = #JOB_2_STEP_01) AND "Unit1.Em6.ControlNodes".utility.sequence.status.seqActive;
   "Unit1.Em6.ControlNodes".utility."step".transition1[201] := ("Unit1.Em6.ControlNodes".utility.sequence.status.currentStep = #JOB_2_STEP_01) AND "Unit1.Em6.ControlNodes".utility.sequence.status.seqActive;
   IF ("Unit1.Em6.ControlNodes".utility.sequence.status.currentStep = #JOB_2_STEP_01) AND "Unit1.Em6.ControlNodes".utility.sequence.status.seqActive AND "Unit1.Em6.ControlNodes".utility."step".transition1[201] THEN
       "Unit1.Em6.ControlNodes".utility.sequence.status.nextStep := #JOB_2_STEP_10;
   END_IF;
END_REGION

REGION Network 24: Step[210] : StackTableOutRear X-Axis GearIn
   RUNG wire#powerrail
      { S7_Templates := "SrcType := DInt" } EQ_Contact(in1 := "Unit1.Em6.ControlNodes".utility.sequence.status.currentStep, in2 := #JOB_2_STEP_10)
      Contact( "Unit1.Em6.ControlNodes".utility.sequence.status.seqActive )
      wire#w1
      Coil( "Unit1.Em6.ControlNodes".utility."step".action1[210] )
   END_RUNG
   RUNG wire#w1
      Contact( "Unit1.Em6.ControlNodes".cm.gearIn.stackTableOutRearAxisZ.InSync )
      Coil( "Unit1.Em6.ControlNodes".utility."step".transition1[210] )
   END_RUNG
   RUNG wire#w1
      Contact( "Unit1.Em6.ControlNodes".utility."step".transition1[210] )
      Move(in := #JOB_2_STEP_11, out1 => "Unit1.Em6.ControlNodes".utility.sequence.status.nextStep)
   END_RUNG
   // the same network as SCL:
   "Unit1.Em6.ControlNodes".utility."step".action1[210] := ("Unit1.Em6.ControlNodes".utility.sequence.status.currentStep = #JOB_2_STEP_10) AND "Unit1.Em6.ControlNodes".utility.sequence.status.seqActive;
   "Unit1.Em6.ControlNodes".utility."step".transition1[210] := ("Unit1.Em6.ControlNodes".utility.sequence.status.currentStep = #JOB_2_STEP_10) AND "Unit1.Em6.ControlNodes".utility.sequence.status.seqActive AND "Unit1.Em6.ControlNodes".cm.gearIn.stackTableOutRearAxisZ.InSync;
   IF ("Unit1.Em6.ControlNodes".utility.sequence.status.currentStep = #JOB_2_STEP_10) AND "Unit1.Em6.ControlNodes".utility.sequence.status.seqActive AND "Unit1.Em6.ControlNodes".utility."step".transition1[210] THEN
       "Unit1.Em6.ControlNodes".utility.sequence.status.nextStep := #JOB_2_STEP_11;
   END_IF;
END_REGION

REGION Network 25: Step[211] : StackTableOutRear X-Axis LimitSensor Off
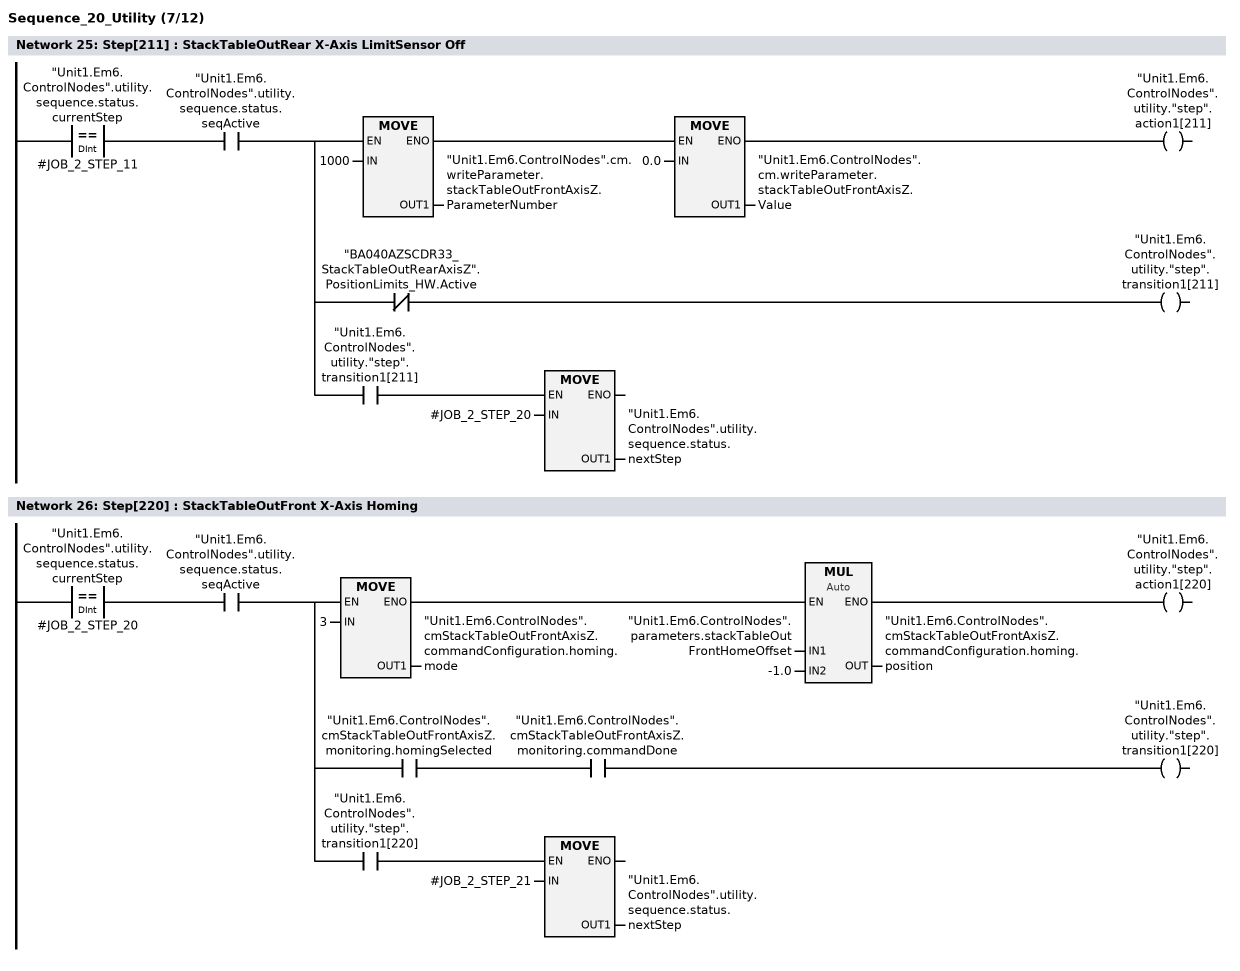
   RUNG wire#powerrail
      { S7_Templates := "SrcType := DInt" } EQ_Contact(in1 := "Unit1.Em6.ControlNodes".utility.sequence.status.currentStep, in2 := #JOB_2_STEP_11)
      Contact( "Unit1.Em6.ControlNodes".utility.sequence.status.seqActive )
      wire#w1
      Move(in := 1000, out1 => "Unit1.Em6.ControlNodes".cm.writeParameter.stackTableOutFrontAxisZ.ParameterNumber)
      Move(in := 0.0, out1 => "Unit1.Em6.ControlNodes".cm.writeParameter.stackTableOutFrontAxisZ.Value)
      Coil( "Unit1.Em6.ControlNodes".utility."step".action1[211] )
   END_RUNG
   RUNG wire#w1
      I_Contact( "BA040AZSCDR33_StackTableOutRearAxisZ".PositionLimits_HW.Active )
      Coil( "Unit1.Em6.ControlNodes".utility."step".transition1[211] )
   END_RUNG
   RUNG wire#w1
      Contact( "Unit1.Em6.ControlNodes".utility."step".transition1[211] )
      Move(in := #JOB_2_STEP_20, out1 => "Unit1.Em6.ControlNodes".utility.sequence.status.nextStep)
   END_RUNG
   // the same network as SCL:
   #_w1 := ("Unit1.Em6.ControlNodes".utility.sequence.status.currentStep = #JOB_2_STEP_11) AND "Unit1.Em6.ControlNodes".utility.sequence.status.seqActive;
   IF #_w1 THEN
       "Unit1.Em6.ControlNodes".cm.writeParameter.stackTableOutFrontAxisZ.ParameterNumber := 1000;
       "Unit1.Em6.ControlNodes".cm.writeParameter.stackTableOutFrontAxisZ.Value := 0.0;
   END_IF;
   "Unit1.Em6.ControlNodes".utility."step".action1[211] := #_w1;
   "Unit1.Em6.ControlNodes".utility."step".transition1[211] := #_w1 AND NOT "BA040AZSCDR33_StackTableOutRearAxisZ".PositionLimits_HW.Active;
   IF #_w1 AND "Unit1.Em6.ControlNodes".utility."step".transition1[211] THEN
       "Unit1.Em6.ControlNodes".utility.sequence.status.nextStep := #JOB_2_STEP_20;
   END_IF;
END_REGION

REGION Network 26: Step[220] : StackTableOutFront X-Axis Homing
   RUNG wire#powerrail
      { S7_Templates := "SrcType := DInt" } EQ_Contact(in1 := "Unit1.Em6.ControlNodes".utility.sequence.status.currentStep, in2 := #JOB_2_STEP_20)
      Contact( "Unit1.Em6.ControlNodes".utility.sequence.status.seqActive )
      wire#w1
      Move(in := 3, out1 => "Unit1.Em6.ControlNodes".cmStackTableOutFrontAxisZ.commandConfiguration.homing.mode)
      Mul(in1 := "Unit1.Em6.ControlNodes".parameters.stackTableOutFrontHomeOffset, in2 := -1.0, out => "Unit1.Em6.ControlNodes".cmStackTableOutFrontAxisZ.commandConfiguration.homing.position)
      Coil( "Unit1.Em6.ControlNodes".utility."step".action1[220] )
   END_RUNG
   RUNG wire#w1
      Contact( "Unit1.Em6.ControlNodes".cmStackTableOutFrontAxisZ.monitoring.homingSelected )
      Contact( "Unit1.Em6.ControlNodes".cmStackTableOutFrontAxisZ.monitoring.commandDone )
      Coil( "Unit1.Em6.ControlNodes".utility."step".transition1[220] )
   END_RUNG
   RUNG wire#w1
      Contact( "Unit1.Em6.ControlNodes".utility."step".transition1[220] )
      Move(in := #JOB_2_STEP_21, out1 => "Unit1.Em6.ControlNodes".utility.sequence.status.nextStep)
   END_RUNG
   // the same network as SCL:
   #_w1 := ("Unit1.Em6.ControlNodes".utility.sequence.status.currentStep = #JOB_2_STEP_20) AND "Unit1.Em6.ControlNodes".utility.sequence.status.seqActive;
   IF #_w1 THEN
       "Unit1.Em6.ControlNodes".cmStackTableOutFrontAxisZ.commandConfiguration.homing.mode := 3;
       "Unit1.Em6.ControlNodes".cmStackTableOutFrontAxisZ.commandConfiguration.homing.position := "Unit1.Em6.ControlNodes".parameters.stackTableOutFrontHomeOffset * (-1.0);
   END_IF;
   "Unit1.Em6.ControlNodes".utility."step".action1[220] := #_w1;
   "Unit1.Em6.ControlNodes".utility."step".transition1[220] := #_w1 AND "Unit1.Em6.ControlNodes".cmStackTableOutFrontAxisZ.monitoring.homingSelected AND "Unit1.Em6.ControlNodes".cmStackTableOutFrontAxisZ.monitoring.commandDone;
   IF #_w1 AND "Unit1.Em6.ControlNodes".utility."step".transition1[220] THEN
       "Unit1.Em6.ControlNodes".utility.sequence.status.nextStep := #JOB_2_STEP_21;
   END_IF;
END_REGION

REGION Network 27: Step[221] : StackTableOutFront X-Axis Move Home
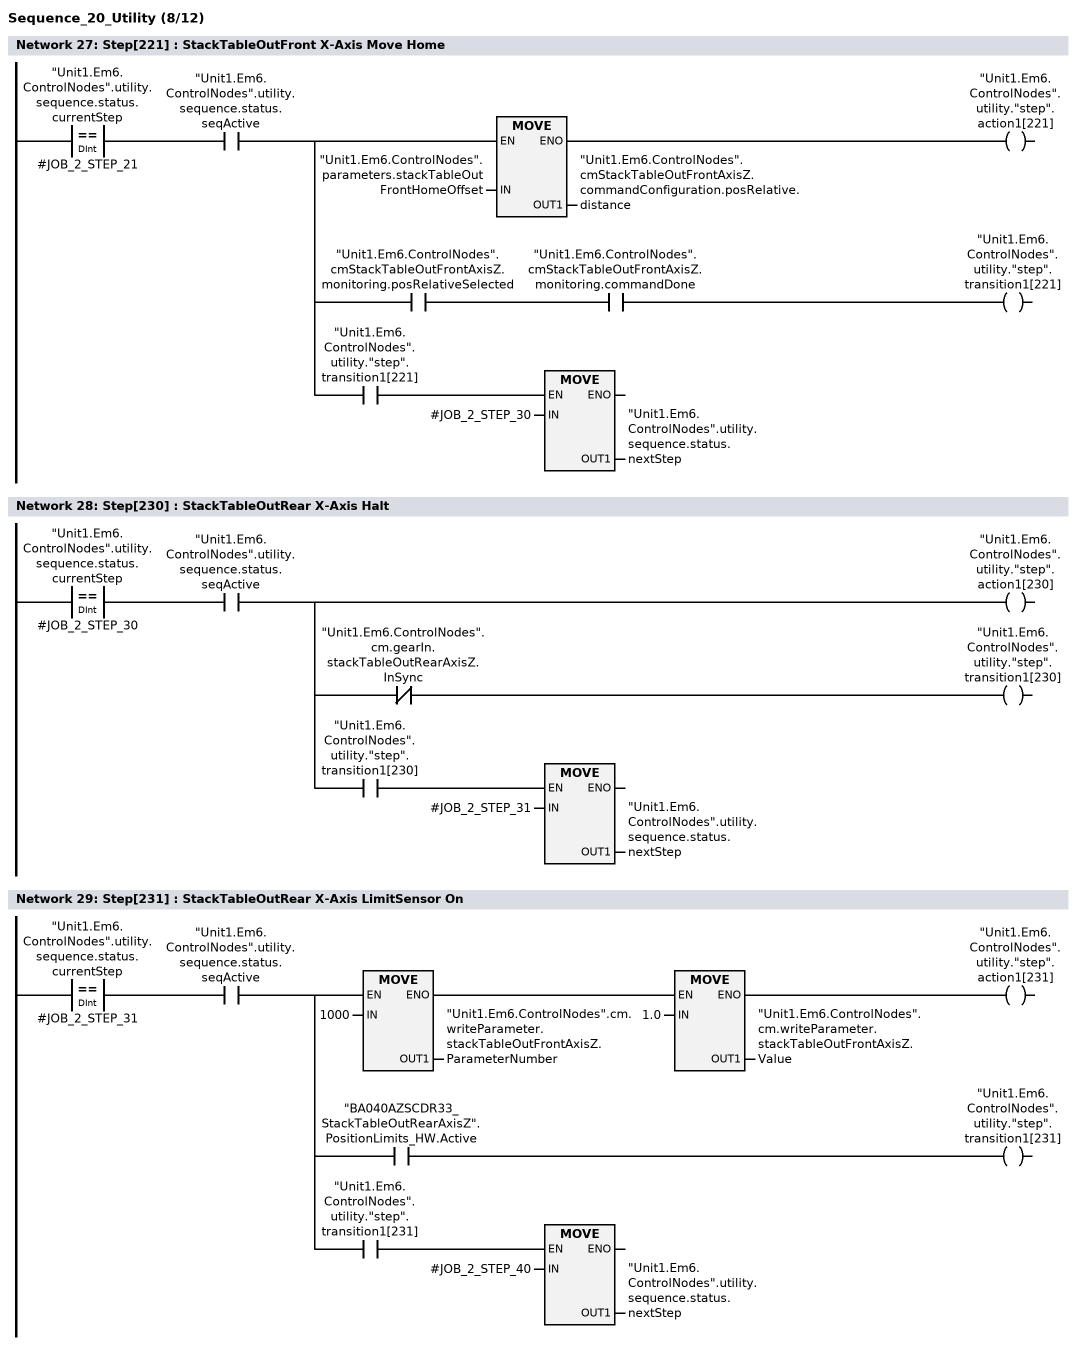
   RUNG wire#powerrail
      { S7_Templates := "SrcType := DInt" } EQ_Contact(in1 := "Unit1.Em6.ControlNodes".utility.sequence.status.currentStep, in2 := #JOB_2_STEP_21)
      Contact( "Unit1.Em6.ControlNodes".utility.sequence.status.seqActive )
      wire#w1
      Move(in := "Unit1.Em6.ControlNodes".parameters.stackTableOutFrontHomeOffset, out1 => "Unit1.Em6.ControlNodes".cmStackTableOutFrontAxisZ.commandConfiguration.posRelative.distance)
      Coil( "Unit1.Em6.ControlNodes".utility."step".action1[221] )
   END_RUNG
   RUNG wire#w1
      Contact( "Unit1.Em6.ControlNodes".cmStackTableOutFrontAxisZ.monitoring.posRelativeSelected )
      Contact( "Unit1.Em6.ControlNodes".cmStackTableOutFrontAxisZ.monitoring.commandDone )
      Coil( "Unit1.Em6.ControlNodes".utility."step".transition1[221] )
   END_RUNG
   RUNG wire#w1
      Contact( "Unit1.Em6.ControlNodes".utility."step".transition1[221] )
      Move(in := #JOB_2_STEP_30, out1 => "Unit1.Em6.ControlNodes".utility.sequence.status.nextStep)
   END_RUNG
   // the same network as SCL:
   #_w1 := ("Unit1.Em6.ControlNodes".utility.sequence.status.currentStep = #JOB_2_STEP_21) AND "Unit1.Em6.ControlNodes".utility.sequence.status.seqActive;
   IF #_w1 THEN
       "Unit1.Em6.ControlNodes".cmStackTableOutFrontAxisZ.commandConfiguration.posRelative.distance := "Unit1.Em6.ControlNodes".parameters.stackTableOutFrontHomeOffset;
   END_IF;
   "Unit1.Em6.ControlNodes".utility."step".action1[221] := #_w1;
   "Unit1.Em6.ControlNodes".utility."step".transition1[221] := #_w1 AND "Unit1.Em6.ControlNodes".cmStackTableOutFrontAxisZ.monitoring.posRelativeSelected AND "Unit1.Em6.ControlNodes".cmStackTableOutFrontAxisZ.monitoring.commandDone;
   IF #_w1 AND "Unit1.Em6.ControlNodes".utility."step".transition1[221] THEN
       "Unit1.Em6.ControlNodes".utility.sequence.status.nextStep := #JOB_2_STEP_30;
   END_IF;
END_REGION

REGION Network 28: Step[230] : StackTableOutRear X-Axis Halt
   RUNG wire#powerrail
      { S7_Templates := "SrcType := DInt" } EQ_Contact(in1 := "Unit1.Em6.ControlNodes".utility.sequence.status.currentStep, in2 := #JOB_2_STEP_30)
      Contact( "Unit1.Em6.ControlNodes".utility.sequence.status.seqActive )
      wire#w1
      Coil( "Unit1.Em6.ControlNodes".utility."step".action1[230] )
   END_RUNG
   RUNG wire#w1
      I_Contact( "Unit1.Em6.ControlNodes".cm.gearIn.stackTableOutRearAxisZ.InSync )
      Coil( "Unit1.Em6.ControlNodes".utility."step".transition1[230] )
   END_RUNG
   RUNG wire#w1
      Contact( "Unit1.Em6.ControlNodes".utility."step".transition1[230] )
      Move(in := #JOB_2_STEP_31, out1 => "Unit1.Em6.ControlNodes".utility.sequence.status.nextStep)
   END_RUNG
   // the same network as SCL:
   "Unit1.Em6.ControlNodes".utility."step".action1[230] := ("Unit1.Em6.ControlNodes".utility.sequence.status.currentStep = #JOB_2_STEP_30) AND "Unit1.Em6.ControlNodes".utility.sequence.status.seqActive;
   "Unit1.Em6.ControlNodes".utility."step".transition1[230] := ("Unit1.Em6.ControlNodes".utility.sequence.status.currentStep = #JOB_2_STEP_30) AND "Unit1.Em6.ControlNodes".utility.sequence.status.seqActive AND NOT "Unit1.Em6.ControlNodes".cm.gearIn.stackTableOutRearAxisZ.InSync;
   IF ("Unit1.Em6.ControlNodes".utility.sequence.status.currentStep = #JOB_2_STEP_30) AND "Unit1.Em6.ControlNodes".utility.sequence.status.seqActive AND "Unit1.Em6.ControlNodes".utility."step".transition1[230] THEN
       "Unit1.Em6.ControlNodes".utility.sequence.status.nextStep := #JOB_2_STEP_31;
   END_IF;
END_REGION

REGION Network 29: Step[231] : StackTableOutRear X-Axis LimitSensor On
   RUNG wire#powerrail
      { S7_Templates := "SrcType := DInt" } EQ_Contact(in1 := "Unit1.Em6.ControlNodes".utility.sequence.status.currentStep, in2 := #JOB_2_STEP_31)
      Contact( "Unit1.Em6.ControlNodes".utility.sequence.status.seqActive )
      wire#w1
      Move(in := 1000, out1 => "Unit1.Em6.ControlNodes".cm.writeParameter.stackTableOutFrontAxisZ.ParameterNumber)
      Move(in := 1.0, out1 => "Unit1.Em6.ControlNodes".cm.writeParameter.stackTableOutFrontAxisZ.Value)
      Coil( "Unit1.Em6.ControlNodes".utility."step".action1[231] )
   END_RUNG
   RUNG wire#w1
      Contact( "BA040AZSCDR33_StackTableOutRearAxisZ".PositionLimits_HW.Active )
      Coil( "Unit1.Em6.ControlNodes".utility."step".transition1[231] )
   END_RUNG
   RUNG wire#w1
      Contact( "Unit1.Em6.ControlNodes".utility."step".transition1[231] )
      Move(in := #JOB_2_STEP_40, out1 => "Unit1.Em6.ControlNodes".utility.sequence.status.nextStep)
   END_RUNG
   // the same network as SCL:
   #_w1 := ("Unit1.Em6.ControlNodes".utility.sequence.status.currentStep = #JOB_2_STEP_31) AND "Unit1.Em6.ControlNodes".utility.sequence.status.seqActive;
   IF #_w1 THEN
       "Unit1.Em6.ControlNodes".cm.writeParameter.stackTableOutFrontAxisZ.ParameterNumber := 1000;
       "Unit1.Em6.ControlNodes".cm.writeParameter.stackTableOutFrontAxisZ.Value := 1.0;
   END_IF;
   "Unit1.Em6.ControlNodes".utility."step".action1[231] := #_w1;
   "Unit1.Em6.ControlNodes".utility."step".transition1[231] := #_w1 AND "BA040AZSCDR33_StackTableOutRearAxisZ".PositionLimits_HW.Active;
   IF #_w1 AND "Unit1.Em6.ControlNodes".utility."step".transition1[231] THEN
       "Unit1.Em6.ControlNodes".utility.sequence.status.nextStep := #JOB_2_STEP_40;
   END_IF;
END_REGION

REGION Network 30: Step[240] : StackTableOutFront X-Axis GearIn
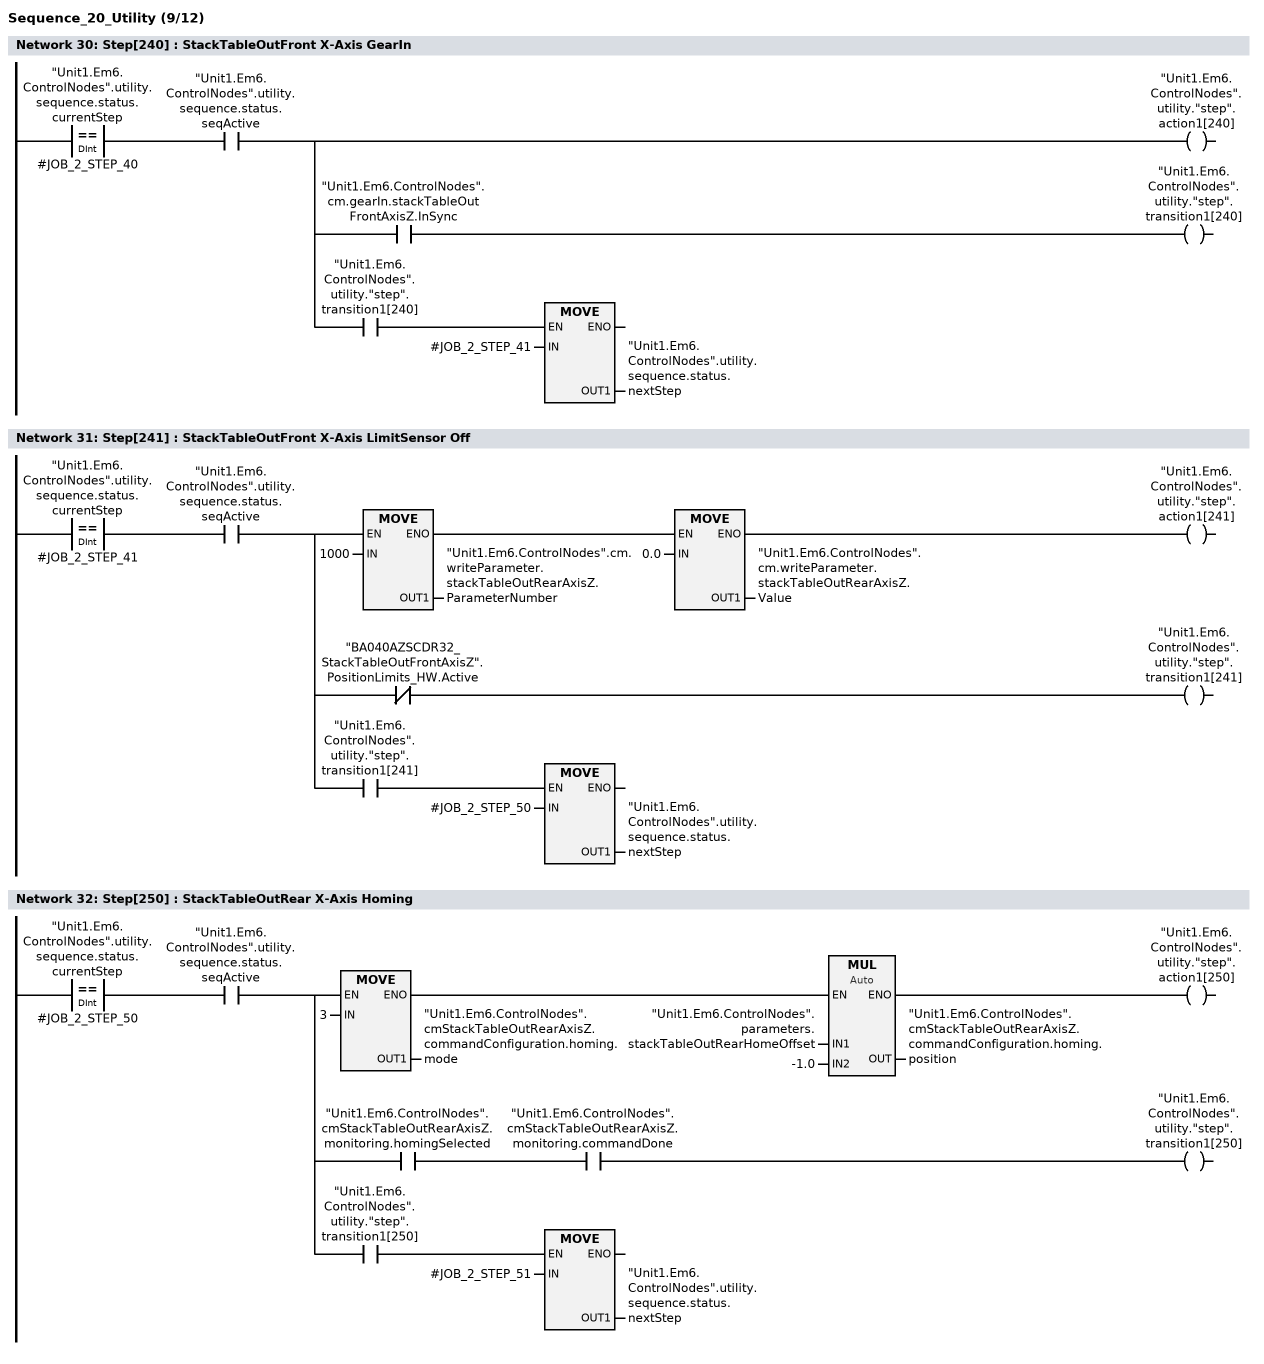
   RUNG wire#powerrail
      { S7_Templates := "SrcType := DInt" } EQ_Contact(in1 := "Unit1.Em6.ControlNodes".utility.sequence.status.currentStep, in2 := #JOB_2_STEP_40)
      Contact( "Unit1.Em6.ControlNodes".utility.sequence.status.seqActive )
      wire#w1
      Coil( "Unit1.Em6.ControlNodes".utility."step".action1[240] )
   END_RUNG
   RUNG wire#w1
      Contact( "Unit1.Em6.ControlNodes".cm.gearIn.stackTableOutFrontAxisZ.InSync )
      Coil( "Unit1.Em6.ControlNodes".utility."step".transition1[240] )
   END_RUNG
   RUNG wire#w1
      Contact( "Unit1.Em6.ControlNodes".utility."step".transition1[240] )
      Move(in := #JOB_2_STEP_41, out1 => "Unit1.Em6.ControlNodes".utility.sequence.status.nextStep)
   END_RUNG
   // the same network as SCL:
   "Unit1.Em6.ControlNodes".utility."step".action1[240] := ("Unit1.Em6.ControlNodes".utility.sequence.status.currentStep = #JOB_2_STEP_40) AND "Unit1.Em6.ControlNodes".utility.sequence.status.seqActive;
   "Unit1.Em6.ControlNodes".utility."step".transition1[240] := ("Unit1.Em6.ControlNodes".utility.sequence.status.currentStep = #JOB_2_STEP_40) AND "Unit1.Em6.ControlNodes".utility.sequence.status.seqActive AND "Unit1.Em6.ControlNodes".cm.gearIn.stackTableOutFrontAxisZ.InSync;
   IF ("Unit1.Em6.ControlNodes".utility.sequence.status.currentStep = #JOB_2_STEP_40) AND "Unit1.Em6.ControlNodes".utility.sequence.status.seqActive AND "Unit1.Em6.ControlNodes".utility."step".transition1[240] THEN
       "Unit1.Em6.ControlNodes".utility.sequence.status.nextStep := #JOB_2_STEP_41;
   END_IF;
END_REGION

REGION Network 31: Step[241] : StackTableOutFront X-Axis LimitSensor Off
   RUNG wire#powerrail
      { S7_Templates := "SrcType := DInt" } EQ_Contact(in1 := "Unit1.Em6.ControlNodes".utility.sequence.status.currentStep, in2 := #JOB_2_STEP_41)
      Contact( "Unit1.Em6.ControlNodes".utility.sequence.status.seqActive )
      wire#w1
      Move(in := 1000, out1 => "Unit1.Em6.ControlNodes".cm.writeParameter.stackTableOutRearAxisZ.ParameterNumber)
      Move(in := 0.0, out1 => "Unit1.Em6.ControlNodes".cm.writeParameter.stackTableOutRearAxisZ.Value)
      Coil( "Unit1.Em6.ControlNodes".utility."step".action1[241] )
   END_RUNG
   RUNG wire#w1
      I_Contact( "BA040AZSCDR32_StackTableOutFrontAxisZ".PositionLimits_HW.Active )
      Coil( "Unit1.Em6.ControlNodes".utility."step".transition1[241] )
   END_RUNG
   RUNG wire#w1
      Contact( "Unit1.Em6.ControlNodes".utility."step".transition1[241] )
      Move(in := #JOB_2_STEP_50, out1 => "Unit1.Em6.ControlNodes".utility.sequence.status.nextStep)
   END_RUNG
   // the same network as SCL:
   #_w1 := ("Unit1.Em6.ControlNodes".utility.sequence.status.currentStep = #JOB_2_STEP_41) AND "Unit1.Em6.ControlNodes".utility.sequence.status.seqActive;
   IF #_w1 THEN
       "Unit1.Em6.ControlNodes".cm.writeParameter.stackTableOutRearAxisZ.ParameterNumber := 1000;
       "Unit1.Em6.ControlNodes".cm.writeParameter.stackTableOutRearAxisZ.Value := 0.0;
   END_IF;
   "Unit1.Em6.ControlNodes".utility."step".action1[241] := #_w1;
   "Unit1.Em6.ControlNodes".utility."step".transition1[241] := #_w1 AND NOT "BA040AZSCDR32_StackTableOutFrontAxisZ".PositionLimits_HW.Active;
   IF #_w1 AND "Unit1.Em6.ControlNodes".utility."step".transition1[241] THEN
       "Unit1.Em6.ControlNodes".utility.sequence.status.nextStep := #JOB_2_STEP_50;
   END_IF;
END_REGION

REGION Network 32: Step[250] : StackTableOutRear X-Axis Homing
   RUNG wire#powerrail
      { S7_Templates := "SrcType := DInt" } EQ_Contact(in1 := "Unit1.Em6.ControlNodes".utility.sequence.status.currentStep, in2 := #JOB_2_STEP_50)
      Contact( "Unit1.Em6.ControlNodes".utility.sequence.status.seqActive )
      wire#w1
      Move(in := 3, out1 => "Unit1.Em6.ControlNodes".cmStackTableOutRearAxisZ.commandConfiguration.homing.mode)
      Mul(in1 := "Unit1.Em6.ControlNodes".parameters.stackTableOutRearHomeOffset, in2 := -1.0, out => "Unit1.Em6.ControlNodes".cmStackTableOutRearAxisZ.commandConfiguration.homing.position)
      Coil( "Unit1.Em6.ControlNodes".utility."step".action1[250] )
   END_RUNG
   RUNG wire#w1
      Contact( "Unit1.Em6.ControlNodes".cmStackTableOutRearAxisZ.monitoring.homingSelected )
      Contact( "Unit1.Em6.ControlNodes".cmStackTableOutRearAxisZ.monitoring.commandDone )
      Coil( "Unit1.Em6.ControlNodes".utility."step".transition1[250] )
   END_RUNG
   RUNG wire#w1
      Contact( "Unit1.Em6.ControlNodes".utility."step".transition1[250] )
      Move(in := #JOB_2_STEP_51, out1 => "Unit1.Em6.ControlNodes".utility.sequence.status.nextStep)
   END_RUNG
   // the same network as SCL:
   #_w1 := ("Unit1.Em6.ControlNodes".utility.sequence.status.currentStep = #JOB_2_STEP_50) AND "Unit1.Em6.ControlNodes".utility.sequence.status.seqActive;
   IF #_w1 THEN
       "Unit1.Em6.ControlNodes".cmStackTableOutRearAxisZ.commandConfiguration.homing.mode := 3;
       "Unit1.Em6.ControlNodes".cmStackTableOutRearAxisZ.commandConfiguration.homing.position := "Unit1.Em6.ControlNodes".parameters.stackTableOutRearHomeOffset * (-1.0);
   END_IF;
   "Unit1.Em6.ControlNodes".utility."step".action1[250] := #_w1;
   "Unit1.Em6.ControlNodes".utility."step".transition1[250] := #_w1 AND "Unit1.Em6.ControlNodes".cmStackTableOutRearAxisZ.monitoring.homingSelected AND "Unit1.Em6.ControlNodes".cmStackTableOutRearAxisZ.monitoring.commandDone;
   IF #_w1 AND "Unit1.Em6.ControlNodes".utility."step".transition1[250] THEN
       "Unit1.Em6.ControlNodes".utility.sequence.status.nextStep := #JOB_2_STEP_51;
   END_IF;
END_REGION

REGION Network 33: Step[251] : StackTableOutRear X-Axis Move Home
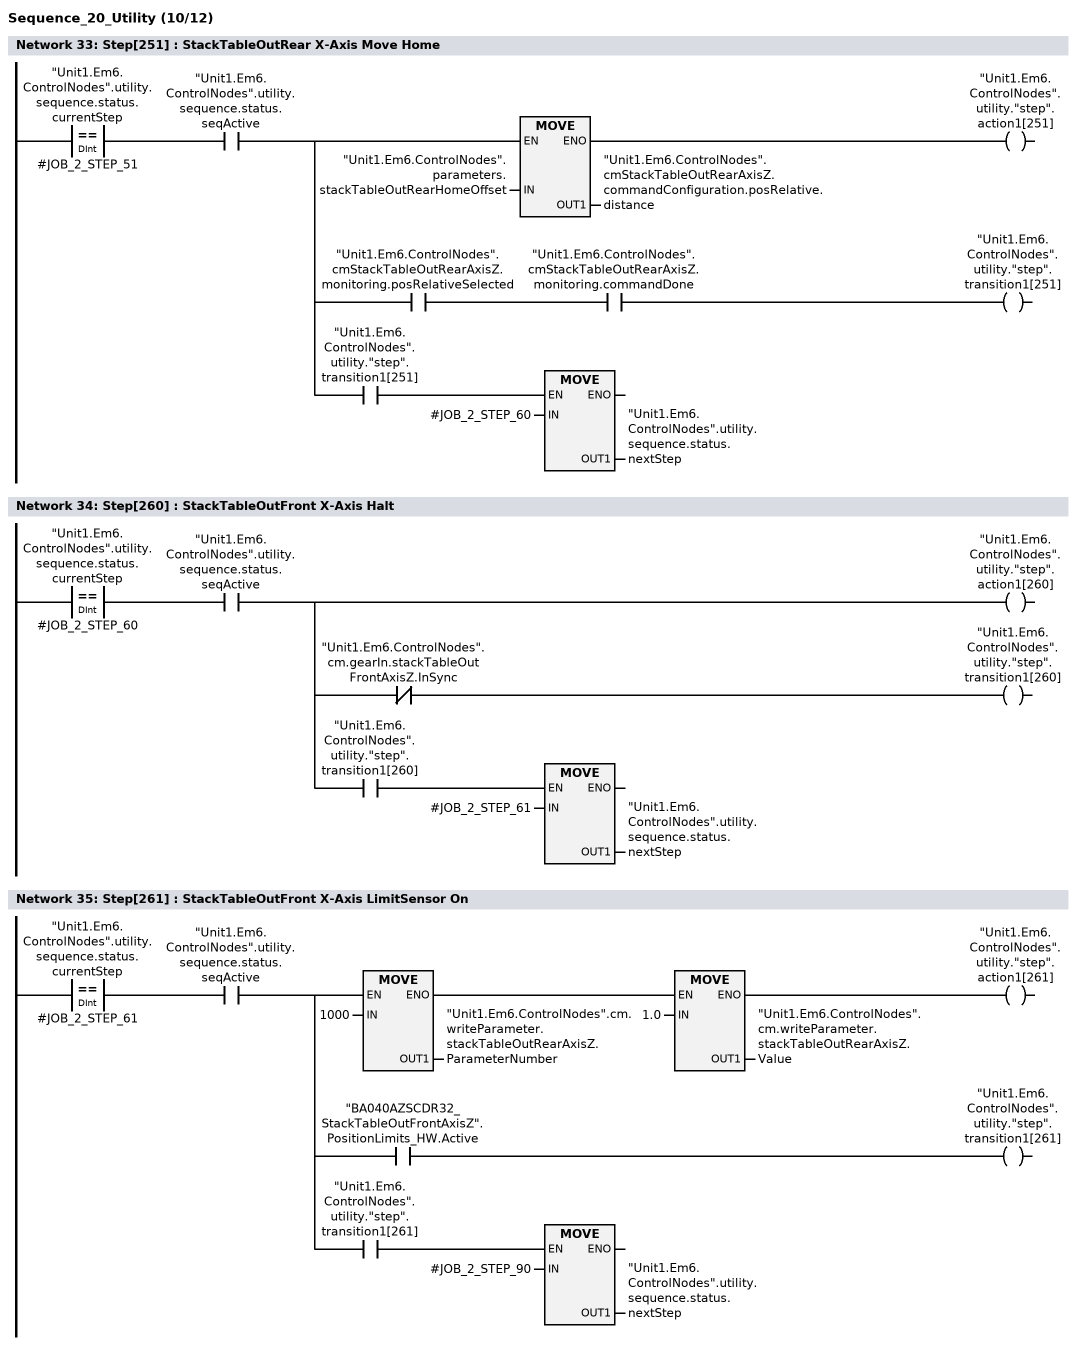
   RUNG wire#powerrail
      { S7_Templates := "SrcType := DInt" } EQ_Contact(in1 := "Unit1.Em6.ControlNodes".utility.sequence.status.currentStep, in2 := #JOB_2_STEP_51)
      Contact( "Unit1.Em6.ControlNodes".utility.sequence.status.seqActive )
      wire#w1
      Move(in := "Unit1.Em6.ControlNodes".parameters.stackTableOutRearHomeOffset, out1 => "Unit1.Em6.ControlNodes".cmStackTableOutRearAxisZ.commandConfiguration.posRelative.distance)
      Coil( "Unit1.Em6.ControlNodes".utility."step".action1[251] )
   END_RUNG
   RUNG wire#w1
      Contact( "Unit1.Em6.ControlNodes".cmStackTableOutRearAxisZ.monitoring.posRelativeSelected )
      Contact( "Unit1.Em6.ControlNodes".cmStackTableOutRearAxisZ.monitoring.commandDone )
      Coil( "Unit1.Em6.ControlNodes".utility."step".transition1[251] )
   END_RUNG
   RUNG wire#w1
      Contact( "Unit1.Em6.ControlNodes".utility."step".transition1[251] )
      Move(in := #JOB_2_STEP_60, out1 => "Unit1.Em6.ControlNodes".utility.sequence.status.nextStep)
   END_RUNG
   // the same network as SCL:
   #_w1 := ("Unit1.Em6.ControlNodes".utility.sequence.status.currentStep = #JOB_2_STEP_51) AND "Unit1.Em6.ControlNodes".utility.sequence.status.seqActive;
   IF #_w1 THEN
       "Unit1.Em6.ControlNodes".cmStackTableOutRearAxisZ.commandConfiguration.posRelative.distance := "Unit1.Em6.ControlNodes".parameters.stackTableOutRearHomeOffset;
   END_IF;
   "Unit1.Em6.ControlNodes".utility."step".action1[251] := #_w1;
   "Unit1.Em6.ControlNodes".utility."step".transition1[251] := #_w1 AND "Unit1.Em6.ControlNodes".cmStackTableOutRearAxisZ.monitoring.posRelativeSelected AND "Unit1.Em6.ControlNodes".cmStackTableOutRearAxisZ.monitoring.commandDone;
   IF #_w1 AND "Unit1.Em6.ControlNodes".utility."step".transition1[251] THEN
       "Unit1.Em6.ControlNodes".utility.sequence.status.nextStep := #JOB_2_STEP_60;
   END_IF;
END_REGION

REGION Network 34: Step[260] : StackTableOutFront X-Axis Halt
   RUNG wire#powerrail
      { S7_Templates := "SrcType := DInt" } EQ_Contact(in1 := "Unit1.Em6.ControlNodes".utility.sequence.status.currentStep, in2 := #JOB_2_STEP_60)
      Contact( "Unit1.Em6.ControlNodes".utility.sequence.status.seqActive )
      wire#w1
      Coil( "Unit1.Em6.ControlNodes".utility."step".action1[260] )
   END_RUNG
   RUNG wire#w1
      I_Contact( "Unit1.Em6.ControlNodes".cm.gearIn.stackTableOutFrontAxisZ.InSync )
      Coil( "Unit1.Em6.ControlNodes".utility."step".transition1[260] )
   END_RUNG
   RUNG wire#w1
      Contact( "Unit1.Em6.ControlNodes".utility."step".transition1[260] )
      Move(in := #JOB_2_STEP_61, out1 => "Unit1.Em6.ControlNodes".utility.sequence.status.nextStep)
   END_RUNG
   // the same network as SCL:
   "Unit1.Em6.ControlNodes".utility."step".action1[260] := ("Unit1.Em6.ControlNodes".utility.sequence.status.currentStep = #JOB_2_STEP_60) AND "Unit1.Em6.ControlNodes".utility.sequence.status.seqActive;
   "Unit1.Em6.ControlNodes".utility."step".transition1[260] := ("Unit1.Em6.ControlNodes".utility.sequence.status.currentStep = #JOB_2_STEP_60) AND "Unit1.Em6.ControlNodes".utility.sequence.status.seqActive AND NOT "Unit1.Em6.ControlNodes".cm.gearIn.stackTableOutFrontAxisZ.InSync;
   IF ("Unit1.Em6.ControlNodes".utility.sequence.status.currentStep = #JOB_2_STEP_60) AND "Unit1.Em6.ControlNodes".utility.sequence.status.seqActive AND "Unit1.Em6.ControlNodes".utility."step".transition1[260] THEN
       "Unit1.Em6.ControlNodes".utility.sequence.status.nextStep := #JOB_2_STEP_61;
   END_IF;
END_REGION

REGION Network 35: Step[261] : StackTableOutFront X-Axis LimitSensor On
   RUNG wire#powerrail
      { S7_Templates := "SrcType := DInt" } EQ_Contact(in1 := "Unit1.Em6.ControlNodes".utility.sequence.status.currentStep, in2 := #JOB_2_STEP_61)
      Contact( "Unit1.Em6.ControlNodes".utility.sequence.status.seqActive )
      wire#w1
      Move(in := 1000, out1 => "Unit1.Em6.ControlNodes".cm.writeParameter.stackTableOutRearAxisZ.ParameterNumber)
      Move(in := 1.0, out1 => "Unit1.Em6.ControlNodes".cm.writeParameter.stackTableOutRearAxisZ.Value)
      Coil( "Unit1.Em6.ControlNodes".utility."step".action1[261] )
   END_RUNG
   RUNG wire#w1
      Contact( "BA040AZSCDR32_StackTableOutFrontAxisZ".PositionLimits_HW.Active )
      Coil( "Unit1.Em6.ControlNodes".utility."step".transition1[261] )
   END_RUNG
   RUNG wire#w1
      Contact( "Unit1.Em6.ControlNodes".utility."step".transition1[261] )
      Move(in := #JOB_2_STEP_90, out1 => "Unit1.Em6.ControlNodes".utility.sequence.status.nextStep)
   END_RUNG
   // the same network as SCL:
   #_w1 := ("Unit1.Em6.ControlNodes".utility.sequence.status.currentStep = #JOB_2_STEP_61) AND "Unit1.Em6.ControlNodes".utility.sequence.status.seqActive;
   IF #_w1 THEN
       "Unit1.Em6.ControlNodes".cm.writeParameter.stackTableOutRearAxisZ.ParameterNumber := 1000;
       "Unit1.Em6.ControlNodes".cm.writeParameter.stackTableOutRearAxisZ.Value := 1.0;
   END_IF;
   "Unit1.Em6.ControlNodes".utility."step".action1[261] := #_w1;
   "Unit1.Em6.ControlNodes".utility."step".transition1[261] := #_w1 AND "BA040AZSCDR32_StackTableOutFrontAxisZ".PositionLimits_HW.Active;
   IF #_w1 AND "Unit1.Em6.ControlNodes".utility."step".transition1[261] THEN
       "Unit1.Em6.ControlNodes".utility.sequence.status.nextStep := #JOB_2_STEP_90;
   END_IF;
END_REGION

REGION Network 36: Step[290] : JOB[2] Step End
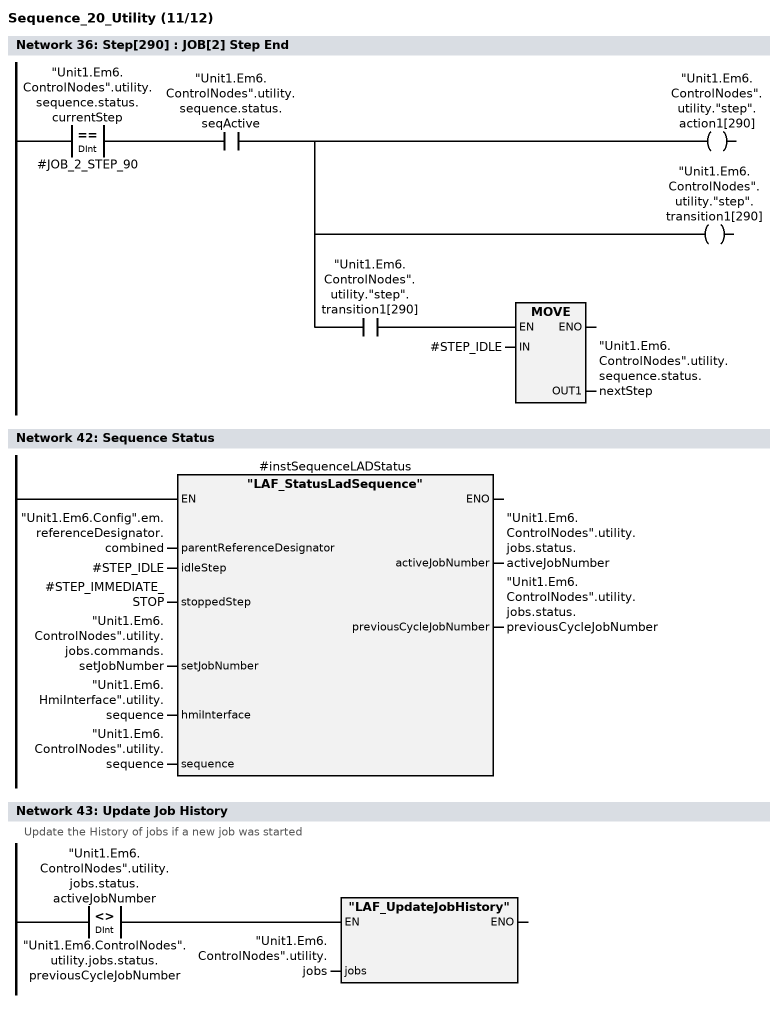
   RUNG wire#powerrail
      { S7_Templates := "SrcType := DInt" } EQ_Contact(in1 := "Unit1.Em6.ControlNodes".utility.sequence.status.currentStep, in2 := #JOB_2_STEP_90)
      Contact( "Unit1.Em6.ControlNodes".utility.sequence.status.seqActive )
      wire#w1
      Coil( "Unit1.Em6.ControlNodes".utility."step".action1[290] )
   END_RUNG
   RUNG wire#w1
      Coil( "Unit1.Em6.ControlNodes".utility."step".transition1[290] )
   END_RUNG
   RUNG wire#w1
      Contact( "Unit1.Em6.ControlNodes".utility."step".transition1[290] )
      Move(in := #STEP_IDLE, out1 => "Unit1.Em6.ControlNodes".utility.sequence.status.nextStep)
   END_RUNG
   // the same network as SCL:
   "Unit1.Em6.ControlNodes".utility."step".action1[290] := ("Unit1.Em6.ControlNodes".utility.sequence.status.currentStep = #JOB_2_STEP_90) AND "Unit1.Em6.ControlNodes".utility.sequence.status.seqActive;
   "Unit1.Em6.ControlNodes".utility."step".transition1[290] := ("Unit1.Em6.ControlNodes".utility.sequence.status.currentStep = #JOB_2_STEP_90) AND "Unit1.Em6.ControlNodes".utility.sequence.status.seqActive;
   IF ("Unit1.Em6.ControlNodes".utility.sequence.status.currentStep = #JOB_2_STEP_90) AND "Unit1.Em6.ControlNodes".utility.sequence.status.seqActive AND "Unit1.Em6.ControlNodes".utility."step".transition1[290] THEN
       "Unit1.Em6.ControlNodes".utility.sequence.status.nextStep := #STEP_IDLE;
   END_IF;
END_REGION

REGION Network 38: *************** IMMEDIATE STOP **************************
END_REGION

REGION Network 39: Immediate Stop
END_REGION

REGION Network 41: *************** Status updates **************************
END_REGION

REGION Network 42: Sequence Status
   RUNG wire#powerrail
      #instSequenceLADStatus(parentReferenceDesignator := "Unit1.Em6.Config".em.referenceDesignator.combined, idleStep := #STEP_IDLE, stoppedStep := #STEP_IMMEDIATE_STOP, setJobNumber := "Unit1.Em6.ControlNodes".utility.jobs.commands.setJobNumber, hmiInterface := "Unit1.Em6.HmiInterface".utility.sequence, sequence := "Unit1.Em6.ControlNodes".utility.sequence, activeJobNumber => "Unit1.Em6.ControlNodes".utility.jobs.status.activeJobNumber, previousCycleJobNumber => "Unit1.Em6.ControlNodes".utility.jobs.status.previousCycleJobNumber)
   END_RUNG
   // the same network as SCL:
   #instSequenceLADStatus(parentReferenceDesignator := "Unit1.Em6.Config".em.referenceDesignator.combined,   // "LAF_StatusLadSequence"
                          idleStep := #STEP_IDLE,
                          stoppedStep := #STEP_IMMEDIATE_STOP,
                          setJobNumber := "Unit1.Em6.ControlNodes".utility.jobs.commands.setJobNumber,
                          hmiInterface := "Unit1.Em6.HmiInterface".utility.sequence,
                          sequence := "Unit1.Em6.ControlNodes".utility.sequence,
                          activeJobNumber => "Unit1.Em6.ControlNodes".utility.jobs.status.activeJobNumber,
                          previousCycleJobNumber => "Unit1.Em6.ControlNodes".utility.jobs.status.previousCycleJobNumber);
END_REGION

REGION Network 43: Update Job History
   // Update the History of jobs if a new job was started
   RUNG wire#powerrail
      { S7_Templates := "SrcType := DInt" } NE_Contact(in1 := "Unit1.Em6.ControlNodes".utility.jobs.status.activeJobNumber, in2 := "Unit1.Em6.ControlNodes".utility.jobs.status.previousCycleJobNumber)
      "LAF_UpdateJobHistory"(jobs := "Unit1.Em6.ControlNodes".utility.jobs)
   END_RUNG
   // the same network as SCL:
   IF "Unit1.Em6.ControlNodes".utility.jobs.status.activeJobNumber <> "Unit1.Em6.ControlNodes".utility.jobs.status.previousCycleJobNumber THEN
       "LAF_UpdateJobHistory"(jobs := "Unit1.Em6.ControlNodes".utility.jobs);
   END_IF;
END_REGION

REGION Network 44: Output steps as String
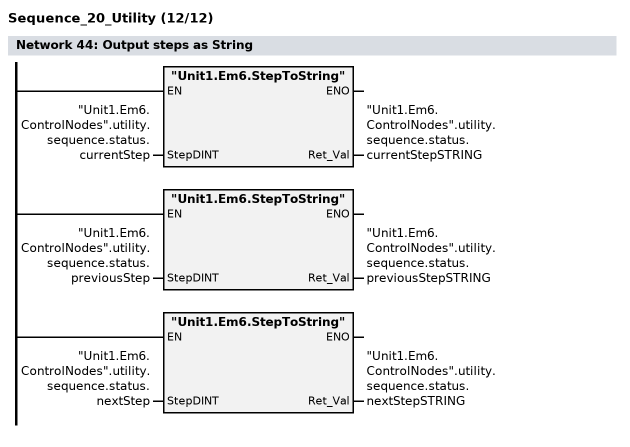
   RUNG wire#powerrail
      "Unit1.Em6.StepToString"(StepDINT := "Unit1.Em6.ControlNodes".utility.sequence.status.currentStep, Ret_Val => "Unit1.Em6.ControlNodes".utility.sequence.status.currentStepSTRING)
   END_RUNG
   RUNG wire#powerrail
      "Unit1.Em6.StepToString"(StepDINT := "Unit1.Em6.ControlNodes".utility.sequence.status.previousStep, Ret_Val => "Unit1.Em6.ControlNodes".utility.sequence.status.previousStepSTRING)
   END_RUNG
   RUNG wire#powerrail
      "Unit1.Em6.StepToString"(StepDINT := "Unit1.Em6.ControlNodes".utility.sequence.status.nextStep, Ret_Val => "Unit1.Em6.ControlNodes".utility.sequence.status.nextStepSTRING)
   END_RUNG
   // the same network as SCL:
   "Unit1.Em6.ControlNodes".utility.sequence.status.currentStepSTRING := "Unit1.Em6.StepToString"(StepDINT := "Unit1.Em6.ControlNodes".utility.sequence.status.currentStep);
   "Unit1.Em6.ControlNodes".utility.sequence.status.previousStepSTRING := "Unit1.Em6.StepToString"(StepDINT := "Unit1.Em6.ControlNodes".utility.sequence.status.previousStep);
   "Unit1.Em6.ControlNodes".utility.sequence.status.nextStepSTRING := "Unit1.Em6.StepToString"(StepDINT := "Unit1.Em6.ControlNodes".utility.sequence.status.nextStep);
END_REGION
END_FUNCTION_BLOCK
